    // ------------------------------------------------------------------
    // ALGORITHM TO PREVIOUS TARGET – TARGET SIDE
    // ------------------------------------------------------------------
    E_RobotState.AlgorithmPreviousTarget:
        yeControl    := RobotControl.vector;
        yinTargetMap := xinMapTarget;
        IF boVectorReached THEN
            eState := E_RobotState.DrivePoint5AlignRFID;//SwitchCoordinatesTarget;
        END_IF
 
    // ------------------------------------------------------------------
    // SWITCH COORDINATES – TARGET SIDE
    // Load target station coordinate from array, switch to position mode.
    // ------------------------------------------------------------------
    E_RobotState.SwitchCoordinatesTarget:
        yeControl                  := RobotControl.position;
		ystTargetPosition.reX      := REAL_TO_LREAL(xarstCoordinates[xinRfidTargetIndex].rePosX) + (crePreTargetDistance * xinTargetDirectionIndex);
        ystTargetPosition.reY      := REAL_TO_LREAL(xarstCoordinates[xinRfidTargetIndex].rePosY);
        ystTargetPosition.reWinkel := REAL_TO_LREAL(xarstCoordinates[xinRfidTargetIndex].reWinkel);
        IF boPositionReached THEN
            eState := E_RobotState.DrivePoint5AlignRFID;
        END_IF
 
    // ------------------------------------------------------------------
    // DRIVE TO POINT 5 – RFID ALIGNMENT POINT + ALIGN
    // Load RFID target coordinate before transitioning.
    // ------------------------------------------------------------------
    E_RobotState.DrivePoint5AlignRFID:
        yeControl := RobotControl.position;
		ystTargetPosition.reX      := REAL_TO_LREAL(xarstCoordinates[xinRfidTargetIndex].rePosX);
        ystTargetPosition.reY      := REAL_TO_LREAL(xarstCoordinates[xinRfidTargetIndex].rePosY);
        ystTargetPosition.reWinkel := REAL_TO_LREAL(xarstCoordinates[xinRfidTargetIndex].reWinkel);
        IF boPositionReached THEN
            eState := E_RobotState.DrivePoint6AtRFID;
        END_IF
 
    // ------------------------------------------------------------------
    // DRIVE TO POINT 6 – AT RFID SENSOR + ALIGN
    // ------------------------------------------------------------------
    E_RobotState.DrivePoint6AtRFID:
        yeControl := RobotControl.position;
        IF TRUE THEN
            eState := E_RobotState.ScanRFIDTarget;
        END_IF
 
    // ------------------------------------------------------------------
    // SCAN RFID – TARGET
    // Signal "waiting for RFID in" to controller. Wait for boRFIDComplete.
    // ------------------------------------------------------------------
    E_RobotState.ScanRFIDTarget:
        yeControl := RobotControl.idle;
        ystMqttOut.sJobState.boWaitForRfidIn := TRUE;
        IF boRfidComplete THEN
            ystMqttOut.sJobState.boWaitForRfidIn := FALSE;
            eState := E_RobotState.DrivePoint5;
        END_IF
 
    // ------------------------------------------------------------------
    // DRIVE TO POINT 5 + ALIGN (return from RFID sensor)
    // ------------------------------------------------------------------
    E_RobotState.DrivePoint5:
		yeControl := RobotControl.vector;
		yboDriveAway := TRUE;
        (*yeControl := RobotControl.position;
		ystTargetPosition.reX      := REAL_TO_LREAL(xarstCoordinates[xinRfidTargetIndex].rePosX) + (crePreTargetDistance * xinTargetDirectionIndex);
        ystTargetPosition.reY      := REAL_TO_LREAL(xarstCoordinates[xinRfidTargetIndex].rePosY);
        ystTargetPosition.reWinkel := REAL_TO_LREAL(xarstCoordinates[xinRfidTargetIndex].reWinkel);*)
        IF xboAwayFromObstacle THEN
			yboDriveAway := FALSE;
            eState := E_RobotState.DrivePoint9Drop;//DrivePoint8BeforeDrop;
        END_IF
 
    // ------------------------------------------------------------------
    // DRIVE TO POINT 8 – BEFORE DROP-OFF
    // ------------------------------------------------------------------
//     E_RobotState.DrivePoint8BeforeDrop:
//         yeControl := RobotControl.position;
// 		ystTargetPosition.reX      := REAL_TO_LREAL(xarstCoordinates[xinTargetIndex].rePosX) + (crePreTargetDistance * xinTargetDirectionIndex);
//         ystTargetPosition.reY      := REAL_TO_LREAL(xarstCoordinates[xinTargetIndex].rePosY);
//         ystTargetPosition.reWinkel := REAL_TO_LREAL(xarstCoordinates[xinTargetIndex].reWinkel);
//         IF boPositionReached THEN
//             eState := E_RobotState.DrivePoint9Drop;
//         END_IF
 
    // ------------------------------------------------------------------
    // DRIVE TO POINT 9 – DROP-OFF POSITION
    // ------------------------------------------------------------------
    E_RobotState.DrivePoint9Drop:
        yeControl := RobotControl.position;
		ystTargetPosition.reX      := REAL_TO_LREAL(xarstCoordinates[xinTargetIndex].rePosX);
        ystTargetPosition.reY      := REAL_TO_LREAL(xarstCoordinates[xinTargetIndex].rePosY);
        ystTargetPosition.reWinkel := REAL_TO_LREAL(xarstCoordinates[xinTargetIndex].reWinkel);
        IF boPositionReached THEN
            eState := E_RobotState.OpenGripper;
        END_IF
 
    // ------------------------------------------------------------------
    // OPEN GRIPPER
    // Wait for workpiece-released confirmation (boWorkpieceLoaded = FALSE).
    // ------------------------------------------------------------------
    E_RobotState.OpenGripper:
        yeControl := RobotControl.idle;
		Gripper.closeGripperCommand := FALSE;

		IF Gripper.state_out = CoreGripperControlState.Open THEN
			ystMqttOut.sJobState.boTransportWorkpiece := FALSE;
			ystMqttOut.sJobState.boWorkpiecePlaced    := TRUE;
			eState := E_RobotState.DrivePoint8AfterDrop;
// 		ELSIF TONGripperTime.Q THEN			// Backup, falls Gripper nicht öffnet	--------------------------------------------------------------------------------------------------------------------------------------Hier einmal
// 			eState := E_RobotState.Standby;	// Hier noch in sinnvolleren Zustand springen
	 	END_IF
 
    // ------------------------------------------------------------------
    // DRIVE TO POINT 8 – RETURN AFTER DROP-OFF
    // ------------------------------------------------------------------
    E_RobotState.DrivePoint8AfterDrop:
		yeControl := RobotControl.vector;
		yboDriveAway := TRUE;
       (* yeControl := RobotControl.position;
		ystTargetPosition.reX      := REAL_TO_LREAL(xarstCoordinates[xinTargetIndex].rePosX) + (crePreTargetDistance * xinTargetDirectionIndex);
        ystTargetPosition.reY      := REAL_TO_LREAL(xarstCoordinates[xinTargetIndex].rePosY);
        ystTargetPosition.reWinkel := REAL_TO_LREAL(xarstCoordinates[xinTargetIndex].reWinkel);
		ystMqttOut.sJobState.boWorkpiecePlaced    := FALSE;*)
        IF xboAwayFromObstacle THEN
			yboDriveAway := FALSE;
            eState := E_RobotState.SelectMapParkPosition;
			 yinTargetMap               := xinMapParking;
        END_IF
 
    // ------------------------------------------------------------------
    // SELECT MAP – PARKING POSITION
    // Start vector algorithm to parking. Output job-done signal.
    // Branch A: new job received while returning → CheckConfirmJob
    // Branch B: normal end                       → Standby
    // ------------------------------------------------------------------
    E_RobotState.SelectMapParkPosition:
		yboPassiveWait := FALSE;
		yboDriveAway := FALSE;
         yinTargetMap               := xinMapParking;
        yeControl                  := RobotControl.vector;
		IF eStateOld <> E_RobotState.DrivePoint1NoWorkpiece THEN
		ystMqttOut.sGeneralState.boReady := TRUE;
		END_IF
		IF xreDistFromGoal > creDistanzForTokenRelease  THEN
			ystMqttOut.sToken.boTokenRelease := TRUE;
		END_IF
        IF boVectorReached THEN
			eState := E_RobotState.Standby;
         ELSIF boNewJob THEN
                eState := E_RobotState.CheckConfirmJob;
		END_IF;
		
END_CASE
 {endregion}

TONTokenRequestTime(IN :=  (E_RobotState.WaitPassiveSource = eState) OR (E_RobotState.WaitpointReachedTarget = eState) ,PT := T#0.2S);
TONGripperTime(IN := (eState = E_RobotState.CloseGripper) OR (E_RobotState.OpenGripper = eState), PT := ctiGripperTime);
TONChargingDelay(IN := boCancelCharging, PT := T#3S);

END_IF
	
	//TEST FÜR PASSIVE WAIT
	//eState := E_RobotState.WaitPassiveTarget;
// ---------------------------------------------------------------------------
// Mirror active state to diagnostic output
// ---------------------------------------------------------------------------
yeCurrentState := eState;
 
{endregion}
{region 'old'}
// ---------------------------------------------------------------------------
// Global control output overrides by state group
// (same pattern as FB_StatesTest – set yeControl after CASE to guarantee
//  correct value regardless of internal state transitions within one scan)
// ---------------------------------------------------------------------------
 (*
// Vector states
IF  (eState = E_RobotState.SelectMapStart)
 OR (eState = E_RobotState.WaitpointReachedSource)
 OR (eState = E_RobotState.AlgorithmPreviousSource)
 OR (eState = E_RobotState.SelectMapTarget)
 OR (eState = E_RobotState.WaitpointReachedTarget)
 OR (eState = E_RobotState.AlgorithmPreviousTarget)
 OR (eState = E_RobotState.SelectMapParkPosition) THEN
    yeControl := RobotControl.vector;
END_IF
 
// Position states
IF  (eState = E_RobotState.SwitchCoordinatesSource)
 OR (eState = E_RobotState.DrivePoint1Align)
 OR (eState = E_RobotState.DrivePoint2Align)
 OR (eState = E_RobotState.AtChargingStation)
 OR (eState = E_RobotState.DrivePoint1AfterCharge)
 OR (eState = E_RobotState.AtStation)
 OR (eState = E_RobotState.DrivePoint1WithWorkpiece)
 OR (eState = E_RobotState.DrivePoint1NoWorkpiece)
 OR (eState = E_RobotState.DrivePoint3Align)
 OR (eState = E_RobotState.DrivePoint4)
 OR (eState = E_RobotState.ScanRFIDSource)
 OR (eState = E_RobotState.DrivePoint3ToTarget)
 OR (eState = E_RobotState.SwitchCoordinatesTarget)
 OR (eState = E_RobotState.DrivePoint5AlignRFID)
 OR (eState = E_RobotState.DrivePoint6AtRFID)
 OR (eState = E_RobotState.ScanRFIDTarget)
 OR (eState = E_RobotState.DrivePoint5)
 OR (eState = E_RobotState.DrivePoint8BeforeDrop)
 OR (eState = E_RobotState.DrivePoint9Drop)
 OR (eState = E_RobotState.DrivePoint8AfterDrop) THEN
    yeControl := RobotControl.position;
END_IF
 
// Idle states
IF  (eState = E_RobotState.LoadMaps)
 OR (eState = E_RobotState.Standby)
 OR (eState = E_RobotState.CloseGripper)
 OR (eState = E_RobotState.OpenGripper)
 OR (eState = E_RobotState.WaitForChargingDone) THEN
    yeControl := RobotControl.idle;
END_IF
 
// Stop states
IF  (eState = E_RobotState.WaitPassiveSource)
 OR (eState = E_RobotState.WaitPassiveTarget) THEN
    yeControl := RobotControl.stop;
END_IF*)
{endregion}

END_FUNCTION_BLOCK

// ---- POUs/HAWinoCore/01_Motors/Gripper.TcPOU
PROGRAM Gripper
VAR_INPUT
	closeGripperCommand		 : BOOL;
	Grippercurrent AT %I* : UINT;
END_VAR
VAR_OUTPUT
	state_out : CoreGripperControlState := CoreGripperControlState.init;
END_VAR
VAR
	state : CoreGripperControlState := CoreGripperControlState.init;
	slider					AT%I* : BOOL;
	partGripped				AT%I* : BOOL;
	
	driveEnable				AT%Q* : BOOL;
	driveVelocity 			AT%Q* : INT;
	current :INT;
	timer : TON;
	
	movementTime : TIME := T#3000MS; //Timevalue for Grippercurrent
END_VAR


current := UINT_TO_INT(Grippercurrent);

CASE state OF
///////////////////////////////////////////////////////////////
 CoreGripperControlState.Init: //Reference opening-drive 
 	state := CoreGripperControlState.opening;
			timer(in := 0, pt:= movementTime); // starts Timer
///////////////////////////////////////////////////////////////		
	CoreGripperControlState.Opening:
		driveEnable:=1;
		driveVelocity:=32767;
		IF current > 50 THEN
			timer(IN:=1);
		END_IF;
		
		IF timer.Q THEN 
			state := CoreGripperControlState.Open;
		END_IF
		state_out := CoreGripperControlState.Opening;
///////////////////////////////////////////////////////////////		
	CoreGripperControlState.Closing:
		driveEnable:=1;
		driveVelocity:=-32767;
		timer(IN:=1);
		IF timer.Q THEN 
			state := CoreGripperControlState.Closed;
		END_IF
		state_out := CoreGripperControlState.Closing;
		
///////////////////////////////////////////////////////////////	
	CoreGripperControlState.Open:	
		driveEnable:=0;
		driveVelocity:=0;
		IF  closeGripperCommand THEN
			state := CoreGripperControlState.Closing;
			timer(in := 0, pt:= movementTime);
		END_IF
		state_out := CoreGripperControlState.Open;
///////////////////////////////////////////////////////////////		
	CoreGripperControlState.Closed:	
		driveEnable:=1;
		driveVelocity:=0;					
		IF NOT closeGripperCommand THEN
			state := CoreGripperControlState.Opening;
			timer(in := 0, pt:= movementTime);
		END_IF
		state_out := CoreGripperControlState.Closed;
		
END_CASE

END_PROGRAM

// ---- POUs/HAWinoCore/05_Bahnplanung/FB_Mapping.TcPOU
FUNCTION_BLOCK FB_Mapping
VAR_INPUT
    xstMqttIn               : sMqttIn;  // Full MQTT input – sJOB.inDestination1/2 are read here
    xinDefaultParkingIndex  : INT;      // Constant parking index (e.g. IDX_PARKING_101)
                                        // passed straight through to output unchanged
END_VAR
 
VAR_OUTPUT
    // --- Indices for FB_RobotStateMachine ---
    yinSourceIndex          : INT;      // xinSourceIndex  of FB_RobotStateMachine
	yinSourceDirectionIndex : INT;      //1 if + and -1 if -
	yinTargetDirectionIndex : INT;      //1 if + and -1 if -
    yinTargetIndex          : INT;      // xinTargetIndex  of FB_RobotStateMachine
    yinRfidSourceIndex      : INT;      // xinRfidSourceIndex
    yinRfidTargetIndex      : INT;      // xinRfidTargetIndex
    yinParkingIndex         : INT;      // xinParkingIndex  (= xinDefaultParkingIndex, passed through)
    yinChargingIndex        : INT;      // xinChargingIndex (only valid when yboJobCharging = TRUE)
    yinMapSource            : INT;      // xinMapSource     (map ID derived from station group)
    yinMapTarget            : INT;      // xinMapTarget     (map ID derived from station group)
 
    // --- Job type flags ---
    yboJobTransport         : BOOL;     // Normal transport job  (D2 ≠ 404)
    yboJobCharging          : BOOL;     // Charging job          (D2 = 404)
    yboDecodeError          : BOOL;     // TRUE if an unknown station number was received
END_VAR
 
VAR
    inDest1                 : INT;      // Local copy of inDestination1
    inDest2                 : INT;      // Local copy of inDestination2
	RobotIndex: INT;
END_VAR

//   Station numbers and their RFID assignments:
//   ┌──────────┬────────────────────────┬───────────────────────────────────┐
//   │ Station  │ Name                   │ Associated RFID index             │
//   ├──────────┼────────────────────────┼───────────────────────────────────┤
//   │  1,  2   │ Storage  (left side)   │ RFID 1 (source) / RFID 2 (target) │
//   │  3,  4   │ Storage  (right side)  │ RFID 2 (source) / RFID 1 (target) │
//   │ 11, 12   │ Production 1+2 left    │ RFID 3 (source) / RFID 4 (target) │
//   │ 21, 22   │ Production 1+2 right   │ RFID 4 (source) / RFID 3 (target) │
//   │ 31, 32   │ Production 3+4 left    │ RFID 5 (source) / RFID 6 (target) │
//   │ 41, 42   │ Production 3+4 right   │ RFID 6 (source) / RFID 5 (target) │
//   │  5,  6   │ Drop-off  (left side)  │ RFID 7 (source) / RFID 8 (target) │
//   │  7,  8   │ Drop-off  (right side) │ RFID 8 (source) / RFID 7 (target) │
//   │201, 202  │ Charging               │ No RFID                            │
//   │101..104  │ Parking (constant)     │ No RFID                            │
//   └──────────┴────────────────────────┴───────────────────────────────────┘
// ---------------------------------------------------------------------------
// Reset outputs each scan
// ---------------------------------------------------------------------------
yinSourceIndex      := 0;
yinTargetIndex      := 0;
yinRfidSourceIndex  := IDX_RFID_1;
yinRfidTargetIndex  := IDX_RFID_1;
yinParkingIndex     := xinDefaultParkingIndex;
yinChargingIndex    := IDX_CHARGING_201;
yinMapSource        := 0;
yinMapTarget        := 0;
yboJobTransport     := FALSE;
yboJobCharging      := FALSE;
yboDecodeError      := FALSE;
 
// ---------------------------------------------------------------------------
// Read destinations from MQTT job struct
// ---------------------------------------------------------------------------
inDest1 := xstMqttIn.sJOB.inDestination1;
inDest2 := xstMqttIn.sJOB.inDestination2;
 
// ---------------------------------------------------------------------------
// Determine job type
// ---------------------------------------------------------------------------
IF inDest2 = 404 THEN
    yboJobCharging  := TRUE;
    yboJobTransport := FALSE;
ELSE
    yboJobCharging  := FALSE;
    yboJobTransport := TRUE;
END_IF
 
// ---------------------------------------------------------------------------
// DECODE SOURCE (Destination 1)
//
// Each station number maps to:
//   - a coordinate array index  (yinSourceIndex)
//   - the RFID index on the SOURCE side of that station (yinRfidSourceIndex)
//   - a map ID for the vector algorithm             (yinMapSource)
// ---------------------------------------------------------------------------
CASE inDest1 OF
 
    // --- Storage – left approach (stations 1, 2) ---
    1:
        yinSourceIndex     := IDX_STORAGE_1;
        yinRfidSourceIndex := IDX_RFID_1;
        yinMapSource       := 1;
		yinSourceDirectionIndex := -1;
 		
    2:
        yinSourceIndex     := IDX_STORAGE_2;
        yinRfidSourceIndex := IDX_RFID_1;
        yinMapSource       := 1;
 		yinSourceDirectionIndex := -1;
    // --- Storage – right approach (stations 3, 4) ---
    3:
        yinSourceIndex     := IDX_STORAGE_3;
        yinRfidSourceIndex := IDX_RFID_2;
        yinMapSource       := 2;
 		yinSourceDirectionIndex := 1;
 
    4:
        yinSourceIndex     := IDX_STORAGE_4;
        yinRfidSourceIndex := IDX_RFID_2;
        yinMapSource       := 2;
  		yinSourceDirectionIndex := 1;
 
    // --- Production 1+2 – left approach (stations 11, 12) ---
    11:
        yinSourceIndex     := IDX_PROD_11;
        yinRfidSourceIndex := IDX_RFID_3;
        yinMapSource       := 3;
 		yinSourceDirectionIndex := -1;
 
    12:
        yinSourceIndex     := IDX_PROD_12;
        yinRfidSourceIndex := IDX_RFID_3;
        yinMapSource       := 3;
 		yinSourceDirectionIndex := -1;
 
    // --- Production 1+2 – right approach (stations 21, 22) ---
    21:
        yinSourceIndex     := IDX_PROD_21;
        yinRfidSourceIndex := IDX_RFID_4;
        yinMapSource       := 4;
  		yinSourceDirectionIndex := 1;
 
    22:
        yinSourceIndex     := IDX_PROD_22;
        yinRfidSourceIndex := IDX_RFID_4;
        yinMapSource       := 4;
  		yinSourceDirectionIndex := 1;
 
    // --- Production 3+4 – left approach (stations 31, 32) ---
    31:
        yinSourceIndex     := IDX_PROD_31;
        yinRfidSourceIndex := IDX_RFID_5;
        yinMapSource       := 5;
 		yinSourceDirectionIndex := -1;
 
    32:
        yinSourceIndex     := IDX_PROD_32;
        yinRfidSourceIndex := IDX_RFID_5;
        yinMapSource       := 5;
 		yinSourceDirectionIndex := -1;
 
    // --- Production 3+4 – right approach (stations 41, 42) ---
    41:
        yinSourceIndex     := IDX_PROD_41;
        yinRfidSourceIndex := IDX_RFID_6;
        yinMapSource       := 6;
  		yinSourceDirectionIndex := 1;
 
    42:
        yinSourceIndex     := IDX_PROD_42;
        yinRfidSourceIndex := IDX_RFID_6;
        yinMapSource       := 6;
  		yinSourceDirectionIndex := 1;
 
    // --- Drop-off – left approach (stations 5, 6) ---
    5:
        yinSourceIndex     := IDX_DROPOFF_5;
        yinRfidSourceIndex := IDX_RFID_7;
        yinMapSource       := 7;
 		yinSourceDirectionIndex := -1;
 
    6:
        yinSourceIndex     := IDX_DROPOFF_6;
        yinRfidSourceIndex := IDX_RFID_7;
        yinMapSource       := 7;
 		yinSourceDirectionIndex := -1;
 
    // --- Drop-off – right approach (stations 7, 8) ---
    7:
        yinSourceIndex     := IDX_DROPOFF_7;
        yinRfidSourceIndex := IDX_RFID_8;
        yinMapSource       := 8;
  		yinSourceDirectionIndex := 1;
 
    8:
        yinSourceIndex     := IDX_DROPOFF_8;
        yinRfidSourceIndex := IDX_RFID_8;
        yinMapSource       := 8;
  		yinSourceDirectionIndex := 1;
 
    // --- Charging stations (Destination1 = charging means the robot should charge) ---
    201:
        yinSourceIndex   := IDX_CHARGING_201;
        yinChargingIndex := IDX_CHARGING_201;
        yinMapSource     := 9;
 
    202:
        yinSourceIndex   := IDX_CHARGING_202;
        yinChargingIndex := IDX_CHARGING_202;
        yinMapSource     := 9;
 
ELSE
    // Unknown station number
    yboDecodeError := TRUE;
 
END_CASE
 
// ---------------------------------------------------------------------------
// DECODE TARGET (Destination 2)
//
// Each station number maps to:
//   - a coordinate array index  (yinTargetIndex)
//   - the RFID index on the TARGET side of that station (yinRfidTargetIndex)
//   - a map ID for the vector algorithm             (yinMapTarget)
//
// Special case: Destination2 = 404 → charging job, no target station needed.
// The RFID on the TARGET side is the opposite side of the same block:
//   left stations  (1,2 / 11,12 / 31,32 / 5,6)  → approached from the right → RFID 2,4,6,8
//   right stations (3,4 / 21,22 / 41,42 / 7,8)  → approached from the left  → RFID 1,3,5,7
// ---------------------------------------------------------------------------
CASE inDest2 OF
 
    // --- Storage – right approach as TARGET (stations 1, 2) ---
    1:
        yinTargetIndex     := IDX_STORAGE_1;
        yinRfidTargetIndex := IDX_RFID_1;
        yinMapTarget       := 1;
  		yinTargetDirectionIndex := -1;
 
    2:
        yinTargetIndex     := IDX_STORAGE_2;
        yinRfidTargetIndex := IDX_RFID_1;
        yinMapTarget       := 1;
   		yinTargetDirectionIndex := -1;
 
    // --- Storage – left approach as TARGET (stations 3, 4) ---
    3:
        yinTargetIndex     := IDX_STORAGE_3;
        yinRfidTargetIndex := IDX_RFID_2;
        yinMapTarget       := 2;
   		yinTargetDirectionIndex := 1;
 
    4:
        yinTargetIndex     := IDX_STORAGE_4;
        yinRfidTargetIndex := IDX_RFID_2;
        yinMapTarget       := 2;
   		yinTargetDirectionIndex := 1;
 
    // --- Production 1+2 – right approach as TARGET (stations 11, 12) ---
    11:
        yinTargetIndex     := IDX_PROD_11;
        yinRfidTargetIndex := IDX_RFID_3;
        yinMapTarget       := 3;
   		yinTargetDirectionIndex := -1;
 
    12:
        yinTargetIndex     := IDX_PROD_12;
        yinRfidTargetIndex := IDX_RFID_3;
        yinMapTarget       := 3;
   		yinTargetDirectionIndex := -1;
 
    // --- Production 1+2 – left approach as TARGET (stations 21, 22) ---
    21:
        yinTargetIndex     := IDX_PROD_21;
        yinRfidTargetIndex := IDX_RFID_4;
        yinMapTarget       := 4;
   		yinTargetDirectionIndex := 1;
 
    22:
        yinTargetIndex     := IDX_PROD_22;
        yinRfidTargetIndex := IDX_RFID_4;
        yinMapTarget       := 4;
   		yinTargetDirectionIndex := 1;
 
    // --- Production 3+4 – right approach as TARGET (stations 31, 32) ---
    31:
        yinTargetIndex     := IDX_PROD_31;
        yinRfidTargetIndex := IDX_RFID_5;
        yinMapTarget       := 5;
   		yinTargetDirectionIndex := -1;
 
    32:
        yinTargetIndex     := IDX_PROD_32;
        yinRfidTargetIndex := IDX_RFID_5;
        yinMapTarget       := 5;
   		yinTargetDirectionIndex := -1;
 
    // --- Production 3+4 – left approach as TARGET (stations 41, 42) ---
    41:
        yinTargetIndex     := IDX_PROD_41;
        yinRfidTargetIndex := IDX_RFID_6;
        yinMapTarget       := 6;
		yinTargetDirectionIndex := 1;
 
    42:
        yinTargetIndex     := IDX_PROD_42;
        yinRfidTargetIndex := IDX_RFID_6;
        yinMapTarget       := 6;
		yinTargetDirectionIndex := 1;
 
    // --- Drop-off – right approach as TARGET (stations 5, 6) ---
    5:
        yinTargetIndex     := IDX_DROPOFF_5;
        yinRfidTargetIndex := IDX_RFID_7;
        yinMapTarget       := 7;
   		yinTargetDirectionIndex := -1;
 
    6:
        yinTargetIndex     := IDX_DROPOFF_6;
        yinRfidTargetIndex := IDX_RFID_7;
        yinMapTarget       := 7;
   		yinTargetDirectionIndex := -1;
 
    // --- Drop-off – left approach as TARGET (stations 7, 8) ---
    7:
        yinTargetIndex     := IDX_DROPOFF_7;
        yinRfidTargetIndex := IDX_RFID_8;
        yinMapTarget       := 8;
   		yinTargetDirectionIndex := 1;
 
    8:
        yinTargetIndex     := IDX_DROPOFF_8;
        yinRfidTargetIndex := IDX_RFID_8;
        yinMapTarget       := 8;
   		yinTargetDirectionIndex := 1;
		
    // --- Special: charging job (Destination2 = 404) ---
    404:
        // Target indices not relevant for charging – leave at default.
        // yboJobCharging is already TRUE from the job-type block above.
        yinTargetIndex     := yinChargingIndex;
        yinRfidTargetIndex := IDX_RFID_1;   // unused for charging
        yinMapTarget       := 9;
 
ELSE
    // Unknown target station number (only flag error if not a charging job)
    IF NOT yboJobCharging THEN
        yboDecodeError := TRUE;
    END_IF
 
END_CASE
 
// ---------------------------------------------------------------------------
// Parking index is always passed through unchanged
// ---------------------------------------------------------------------------
RobotIndex := Var_HAWIno.Robot_Number;
 CASE RobotIndex OF 
	1:yinParkingIndex := IDX_PARKING_101;
	2:yinParkingIndex := IDX_PARKING_102;
	3:yinParkingIndex := IDX_PARKING_103;
	4:yinParkingIndex := IDX_PARKING_104;
END_CASE

END_FUNCTION_BLOCK

// ---- POUs/HAWinoCore/05_Bahnplanung/FB_MQTT.TcPOU
FUNCTION_BLOCK FB_MQTT
VAR
    fbClient        : FB_IotMqttClient;
    fbMessageQueue  : FB_IotMqttMessageQueue;
    fbMessage       : FB_IotMqttMessage;
    bSubscribed     : BOOL;
    sReceived       : STRING;
    bSendError   : BOOL;
	bSendJob	:	BOOL;
	bSendState	: BOOL;
	bSendToken	: BOOL;
    sReceivedjob	: STRING(1000);
	sReceivedcmd 	: STRING(1000);
	sSendError    : STRING(1000);
	sSendJob    : STRING(1000);
	sSendState    : STRING := 'State';
	sSendToken    : STRING := 'Token';
	sMqttSEND : sMqttOut;
	sMqttRECEIVE : sMqttIn;
	sSendCharging : STRING;
	
	//Alten Strings speichern
	tempsSendError : STRING(1000);
	tempsSendJob : STRING(1000);
	tempsSendState : STRING(1000);
	tempsSendToken : STRING(1000);
	
	    // JSON Parser
    fbJson          : FB_JsonDomParser;
    jsonDoc         : SJsonValue;
    jsonNode        : SJsonValue;
    
    // Parsed Variablen Empfangen
    boStop          : BOOL;
    boReset         : BOOL;
    boJobReset      : BOOL;
	boRfidComplete	: BOOL;
	boStartJob		: BOOL;
	boTokenGrant	: BOOL;
	boCancelCharging: BOOL;
	
	// Parsed Variablen Senden
	boErrorRoutePlanning: BOOL := FALSE;
	boErrorControl		: BOOL := FALSE;
	boErrorNoWorkpiece	:BOOL := FALSE;
	boErrorWorkpieceLost: BOOL := FALSE;
	
	//Brauchte ne VAR
	charging_dock : INT;
	loading_speed : INT;
	sSendStop : STRING;
	tempjob : STRING;
	tempcmd : STRING;
	tempserror : STRING;
	tempsjob : STRING;
	tempsstate : STRING;
	tempstoken : STRING;
	start : BOOL;
	sReceivedStart : STRING;
	LADEN : BOOL;
	TONPosition : TON;
	boTONFlanke : BOOL;
	tempInit : STRING;
	temprToken : STRING;
	sReceivedToken : STRING;
	station_id : STRING;
	
END_VAR

VAR_INPUT
	xsDataToSend : sMqttOut;
	xsKoordinate : sKoordinate;
	xinMqttTokenTargetId : INT;
END_VAR
VAR_OUTPUT
	ysDataToReceive : sMqttIn;
END_VAR

// Verbindungsparameter setzen

fbClient.sHostName	:=	'192.168.0.11';
fbClient.nHostPort	:= 	1883;
fbClient.sUserName	:=	'VPJ';
fbClient.sUserPassword	:=	'R462';

// Queue mit Client verknüpfen
fbClient.ipMessageQueue := fbMessageQueue;
fbClient.Execute(bConnect := TRUE);

sMqttSEND := xsDataToSend;

// Einmalig subscriben wenn verbunden
IF fbClient.bConnected AND NOT bSubscribed THEN
	tempjob := CONCAT('HAWino/', INT_TO_STRING(Robot_Number));
	tempjob := CONCAT(tempjob, '/job');
    fbClient.Subscribe(
        sTopic := tempjob,
        eQoS   := 0
    );
	tempcmd := CONCAT('HAWino/', INT_TO_STRING(Robot_Number));
	tempcmd := CONCAT(tempcmd, '/cmd');
	fbClient.Subscribe(
        sTopic := tempcmd,
        eQoS   := 0
    );
	
	tempInit := CONCAT('HAWino/', INT_TO_STRING(Robot_Number));
	tempInit := CONCAT(tempInit, '/init');
	fbClient.Subscribe(
        sTopic := tempInit,
        eQoS   := 0
    );
	
	temprToken := CONCAT('HAWino/', INT_TO_STRING(Robot_Number));
	temprToken := CONCAT(temprToken, '/token');
	fbClient.Subscribe(
        sTopic := temprToken,
        eQoS   := 0
    );
	
	tempserror := CONCAT('HAWino/', INT_TO_STRING(Robot_Number));
	tempserror := CONCAT(tempserror, '/error');
	
	tempsjob := CONCAT('HAWino/', INT_TO_STRING(Robot_Number));
	tempsjob := CONCAT(tempsjob, '/jobState');
	
	tempsstate := CONCAT('HAWino/', INT_TO_STRING(Robot_Number));
	tempsstate := CONCAT(tempsstate, '/generalState');
	
// 	tempstoken := CONCAT('agents/station/test_station/token', INT_TO_STRING(Robot_Number));
// 	tempstoken := CONCAT(tempstoken, '/token');
	
	bSubscribed := TRUE;
END_IF

// Nachrichten aus Queue lesen
IF fbMessageQueue.nQueuedMessages > 0 THEN
    fbMessageQueue.Dequeue(fbMessage := fbMessage);
    fbMessage.GetPayload(
        pPayload             := ADR(sReceived),
        nPayloadSize         := SIZEOF(sReceived),
        bSetNullTermination  := TRUE
    );
	    IF fbMessage.CompareTopic(sTopic := tempjob) THEN
        fbMessage.GetPayload(pPayload := ADR(sReceivedjob), nPayloadSize := SIZEOF(sReceivedjob), bSetNullTermination := TRUE);
    
    	ELSIF fbMessage.CompareTopic(sTopic := tempcmd) THEN
        fbMessage.GetPayload(pPayload := ADR(sReceivedcmd), nPayloadSize := SIZEOF(sReceivedcmd), bSetNullTermination := TRUE);
		
 		ELSIF fbMessage.CompareTopic(sTopic := tempInit) THEN
         fbMessage.GetPayload(pPayload := ADR(sReceivedStart), nPayloadSize := SIZEOF(sReceivedStart), bSetNullTermination := TRUE);
 		ELSIF fbMessage.CompareTopic(sTopic := temprToken) THEN
         fbMessage.GetPayload(pPayload := ADR(sReceivedToken), nPayloadSize := SIZEOF(sReceivedToken), bSetNullTermination := TRUE);
		END_IF
	
// Start Parsen
    // jsonDoc := fbJson.ParseDocument(sReceivedStart);
	
  (*   IF jsonDoc <> 0 THEN
         // Init auslesen
        jsonNode := fbJson.FindMember(jsonDoc, 'test');
         IF jsonNode <> 0 THEN
             start := fbJson.GetString(jsonNode) = 'TRUE';
         END_IF
	*)
	
	// JSON parsen CMD
    jsonDoc := fbJson.ParseDocument(sReceivedcmd);
    
    IF jsonDoc <> 0 THEN
        // boStop auslesen
        jsonNode := fbJson.FindMember(jsonDoc, 'boStop');
        IF jsonNode <> 0 THEN
            sMqttRECEIVE.sCmd.boStop := fbJson.GetBool(jsonNode);
        END_IF
        
        // boReset auslesen
        jsonNode := fbJson.FindMember(jsonDoc, 'boReset');
        IF jsonNode <> 0 THEN
            sMqttRECEIVE.sCmd.boReset := fbJson.GetBool(jsonNode);
        END_IF
        
        // boJobReset auslesen
        jsonNode := fbJson.FindMember(jsonDoc, 'boJobReset');
        IF jsonNode <> 0 THEN
            sMqttRECEIVE.sCmd.boJobReset := fbJson.GetBool(jsonNode);
        END_IF
		
		// boRfidComplete auslesen
        jsonNode := fbJson.FindMember(jsonDoc, 'boRfidComplete');
        IF jsonNode <> 0 THEN
            sMqttRECEIVE.sCmd.boRFIDComplete := fbJson.GetBool(jsonNode);
        END_IF
		
		// boStartJob auslesen
        jsonNode := fbJson.FindMember(jsonDoc, 'boStartJob');
        IF jsonNode <> 0 THEN
            sMqttRECEIVE.sCmd.boStartJob := fbJson.GetBool(jsonNode);
        END_IF
		
// 		// boTokenGrant auslesen
//         jsonNode := fbJson.FindMember(jsonDoc, 'boTokenGrant');
//         IF jsonNode <> 0 THEN
//             sMqttRECEIVE.sCmd.boTokenGrant := fbJson.GetString(jsonNode) = 'TRUE';
//         END_IF
		
		// boCancelCharging auslesen
        jsonNode := fbJson.FindMember(jsonDoc, 'boCancelCharging');
        IF jsonNode <> 0 THEN
            sMqttRECEIVE.sCmd.boCancelCharging := fbJson.GetBool(jsonNode);
        END_IF
    END_IF
	
	// JSON parsen CMD
    jsonDoc := fbJson.ParseDocument(sReceivedjob);
	
    IF jsonDoc <> 0 THEN
        // JobID auslesen
        jsonNode := fbJson.FindMember(jsonDoc, 'jobId');
        IF jsonNode <> 0 THEN
            sMqttRECEIVE.sJOB.inJobID := DINT_TO_INT(fbJson.GetInt(jsonNode));
        END_IF
        
        // Destination 1 auslesen
        jsonNode := fbJson.FindMember(jsonDoc, 'inDestination1');
        IF jsonNode <> 0 THEN
            sMqttRECEIVE.sJOB.inDestination1 := DINT_TO_INT(fbJson.GetInt(jsonNode));
        END_IF
        
        // Destination 2 auslesen
        jsonNode := fbJson.FindMember(jsonDoc, 'inDestination2');
        IF jsonNode <> 0 THEN
            sMqttRECEIVE.sJOB.inDestination2 := DINT_TO_INT(fbJson.GetInt(jsonNode));
        END_IF
    END_IF
	
	// JSON parsen Token
    jsonDoc := fbJson.ParseDocument(sReceivedToken);
    IF jsonDoc <> 0 THEN
        // Token Granted auslesen
		jsonNode := fbJson.FindMember(jsonDoc, 'category');
		IF jsonNode <> 0 THEN
			IF fbJson.GetString(jsonNode) = 'TOKEN_GRANT' THEN
				sMqttRECEIVE.sCmd.boTokenGrant := TRUE;
			END_IF
		END_IF
    END_IF
END_IF

start := TRUE;

IF start THEN
	// Die gesendeten Strings abspeichern
	tempsSendError := sSendError;
	tempsSendJob := sSendJob;
	tempsSendState := sSendState;
	tempsSendToken := sSendToken;
	
	
	// Kompletten Error-JSON zusammenbauen
	sSendError := CONCAT('{"boErrorRoutePlanning":"', BOOL_TO_STRING(sMqttSEND.sError.boErrorRoutePlanning));
	sSendError := CONCAT(sSendError, '","boErrorControl":"');
	sSendError := CONCAT(sSendError, BOOL_TO_STRING(sMqttSEND.sError.boErrorControl));
	sSendError := CONCAT(sSendError, '","boErrorNoWorkpiece":"');
	sSendError := CONCAT(sSendError, BOOL_TO_STRING(sMqttSEND.sError.boErrorNoWorkpiece));
	sSendError := CONCAT(sSendError, '","boErrorWorkpieceLost":"');
	sSendError := CONCAT(sSendError, BOOL_TO_STRING(sMqttSEND.sError.boErrorWorkpieceLost));
	sSendError := CONCAT(sSendError, '"}');
	
	// Kompletten jobState-JSON zusammenbauen
	sSendJob := CONCAT('{"boWorkpieceLoaded":"', BOOL_TO_STRING(sMqttSEND.sJobState.boWorkpieceLoaded));
	sSendJob := CONCAT(sSendJob, '","boTransportWorkpiece":"');
	sSendJob := CONCAT(sSendJob, BOOL_TO_STRING(sMqttSEND.sJobState.boTransportWorkpiece));
	sSendJob := CONCAT(sSendJob, '","boJobAccepted":"');
	sSendJob := CONCAT(sSendJob, BOOL_TO_STRING(sMqttSEND.sJobState.boJobAccepted));
	sSendJob := CONCAT(sSendJob, '","boWaitForRfidOut":"');
	sSendJob := CONCAT(sSendJob, BOOL_TO_STRING(sMqttSEND.sJobState.boWaitForRfidOut));
	sSendJob := CONCAT(sSendJob, '","boWaitForRfidIn":"');
	sSendJob := CONCAT(sSendJob, BOOL_TO_STRING(sMqttSEND.sJobState.boWaitForRfidIn));
	sSendJob := CONCAT(sSendJob, '","boWorkpiecePlaced":"');
	sSendJob := CONCAT(sSendJob, BOOL_TO_STRING(sMqttSEND.sJobState.boWorkpiecePlaced));
	sSendJob := CONCAT(sSendJob, '"}');
	
	
	sMqttSEND.sGeneralState.strPosition := CONCAT(CONCAT(REAL_TO_STRING(xsKoordinate.rePosX),','),REAL_TO_STRING(xsKoordinate.rePosY));
	
	// Kompletten generalState-JSON zusammenbauen
	sSendState := CONCAT('{"boReady":"', BOOL_TO_STRING(sMqttSEND.sGeneralState.boReady));
	sSendState := CONCAT(sSendState, '","boCharging":"');
	sSendState := CONCAT(sSendState, BOOL_TO_STRING(sMqttSEND.sGeneralState.boCharging));
	sSendState := CONCAT(sSendState, '","strPosition":"');
	sSendState := CONCAT(sSendState, sMqttSEND.sGeneralState.strPosition);
	sSendState := CONCAT(sSendState, '"}');
	
	// Kompletten Token-JSON
	IF sMqttSEND.sToken.boTokenRequest THEN
		sSendToken := CONCAT('{"category":"TOKEN_REQUEST","robot_id":"', INT_TO_STRING(Robot_Number));
		sSendToken := CONCAT(sSendToken, '"}');
	END_IF
	IF sMqttSEND.sToken.boTokenRelease THEN
		sSendToken := CONCAT('{"category":"TOKEN_RELEASE","robot_id":"', INT_TO_STRING(Robot_Number));
		sSendToken := CONCAT(sSendToken, '"}');
	END_IF
	
	//Charging Request
	sSendCharging := CONCAT('{"robot":"', INT_TO_STRING(Robot_Number));
	sSendCharging := CONCAT(sSendCharging, '","charge":"true');
	sSendCharging := CONCAT(sSendCharging, '","charging_dock":"');
	sSendCharging := CONCAT(sSendCharging, INT_TO_STRING(charging_dock));
	sSendCharging := CONCAT(sSendCharging, '","loading_speed":"');
	sSendCharging := CONCAT(sSendCharging, INT_TO_STRING(loading_speed));
	sSendCharging := CONCAT(sSendCharging, '"}');
	
	//Aufladen stoppen
	sSendStop := CONCAT('{"robot":"', INT_TO_STRING(Robot_Number));
	sSendStop := CONCAT(sSendStop, '","charge":"false');
	sSendStop := CONCAT(sSendStop, '","charging_dock":"');
	sSendStop := CONCAT(sSendStop, INT_TO_STRING(charging_dock));
	sSendStop := CONCAT(sSendStop, '","loading_speed":"');
	sSendStop := CONCAT(sSendStop, INT_TO_STRING(loading_speed));
	sSendStop := CONCAT(sSendStop, '"}');
	
	
	
	// Nur senden wenn sich etwas geändert hat
	IF tempsSendError <> sSendError THEN
		bSendError := TRUE;
	END_IF
	IF tempsSendJob <> sSendJob THEN
		bSendJob := TRUE;
	END_IF

	
	TONPosition(IN := NOT boTONFlanke ,PT := T#0.5S);
	boTONFlanke := TONPOsition.Q;	
	
	IF boTONFlanke THEN
		bSendState := TRUE;
	END_IF

	IF tempsSendToken <> sSendToken THEN
		bSendToken := TRUE;
	END_IF
	
	
	IF fbClient.bConnected THEN
		IF bSendError THEN
			fbClient.Publish(
				sTopic       := tempserror,
				pPayload     := ADR(sSendError),
				nPayloadSize := LEN(sSendError),
				eQoS         := 0,
				bRetain      := FALSE,
				bQueue       := FALSE
			);
			bSendError := FALSE;
		END_IF
	
		IF bSendJob THEN
			fbClient.Publish(
				sTopic       := tempsjob,
				pPayload     := ADR(sSendJob),
				nPayloadSize := LEN(sSendJob),
				eQoS         := 0,
				bRetain      := FALSE,
				bQueue       := FALSE
			);
			bSendJob := FALSE;
		END_IF
	
		IF bSendState THEN
			fbClient.Publish(
				sTopic       := tempsstate,
				pPayload     := ADR(sSendState),
				nPayloadSize := LEN(sSendState),
				eQoS         := 0,
				bRetain      := FALSE,
				bQueue       := FALSE
			);
			bSendState := FALSE;
		END_IF
	
	CASE xinMqttTokenTargetId OF
		1: station_id := 'storage_1';
		2: station_id := 'manufacturing_1';
		3: station_id := 'manufacturing_3';
		4: station_id := 'manufacturing_3';
		5: station_id := 'dispatch';
		
	END_CASE
	tempstoken := CONCAT('agents/station/', station_id); 
	tempstoken := CONCAT(tempstoken,'/token');
		IF bSendToken THEN
			fbClient.Publish(
				sTopic       := tempstoken,
				pPayload     := ADR(sSendToken),
				nPayloadSize := LEN(sSendToken),
				eQoS         := 0,
				bRetain      := FALSE,
				bQueue       := FALSE
			);
			bSendToken := FALSE;
		END_IF
// 		// Roboter will Laden
//  		IF NOT LADEN THEN
//   			fbClient.Publish(
//   				sTopic       := 'ChargingRequest',
//   				pPayload     := ADR(sSendCharging),
//   				nPayloadSize := LEN(sSendCharging),
//   				eQoS         := 0,
//   				bRetain      := FALSE,
//   				bQueue       := FALSE
//   			);
// 			LADEN		 := TRUE;
//  		END_IF
// 		//Roboter soll laden beenden
// 		IF boCancelCharging = TRUE AND E_RobotState = 8 THEN
// 			fbClient.Publish(
// 				sTopic       := 'ChargingRequest',
// 				pPayload     := ADR(sSendStop),
// 				nPayloadSize := LEN(sSendStop),
// 				eQoS         := 0,
// 				bRetain      := FALSE,
// 				bQueue       := FALSE
// 			);
// 		END_IF
	END_IF
END_IF

ysDataToReceive := sMqttRECEIVE;

END_FUNCTION_BLOCK

// ---- POUs/HAWinoCore/HAWino.TcPOU
PROGRAM HAWino
VAR
	Robot_Number	AT%Q*	: INT;
	operationState : DUT_SysState := DUT_SysState.init; 
	RobotData : RobotInternalData;
	GetId : Tc2_Utilities.FB_GetSystemId;
	init : INT;
	SysGUID : GUID;
	start : BOOL:= TRUE;
	
	// Outputs
	initDone AT%Q* : BOOL := FALSE;
	cameraPosition AT%Q* : Position := (x := 0.0, y := 0.0, theta := 0.0, e := 0.0);	// Aktuelle roboterspezifische Kameraposition
	cameraReceivedPakets AT%Q* : UINT;													// Counter für erhaltene Kamerapakete
END_VAR

CASE operationState OF
	//Get SysId for Identification
	DUT_SysState.init:
		GetId(bexecute := start,stSystemId=>SysGUID);
		IF NOT GetId.bBusy THEN	
			operationState:=DUT_SysState.preOp;
		END_IF
	DUT_SysState.preOp:
	//Set RobotNumber for MQTT and set flag to start MQTT
		IF InitSysId(GUID_to_String(SysGUID)) THEN
			Var_HAWIno.Robot_Number := RobotData.Robot_Number;		
			initDone := TRUE;
			operationState:=DUT_SysState.Op;
		END_IF
	DUT_SysState.Op:
	//Operate System

		MQTT();
		IrDistanceSensors();
		Camera();
		cameraPosition := Camera.cameraData.robotPosition[RobotData.Robot_Number]; //Zuweisung der roboterspezifischen Kameraposition
		cameraReceivedPakets := Camera.cameraData.nReceivedPakets;	// Zuweisung der Anzahl der vom Kamerasystem versendeten Pakete (Ueberwachungszwecke)
END_CASE

METHOD InitSysId : BOOL
VAR_INPUT
	SysId : STRING;
END_VAR
VAR
	state : INT;
	CX31C9D6 : STRING := '77726FC0-DD5E-F7D7-002E-41ED9B95AABA';
	CX35CFB8 : STRING := '2A7FC16A-555A-D05D-0E28-E804E05477FE';
	CX35CDC8 : STRING := 'AD3D576A-9CE4-FB95-7439-909C21AA2B33';
	CX35CDD6 : STRING := '975A6B25-37E2-0E46-4C4D-43CCC26F2A66';
	CX4D0046 : STRING := '4FFA7061-8E1F-E1C9-731A-38EAA9BAEAC6';
END_VAR
// CX-31C9D6 = 1
// CX-35CFB8 = 2
// CX-35CDC8 = 3
// CX-35CDD6 = 4
// CX-4D0046 = 5
IF SysId = CX31C9D6 THEN
	state := 1;
ELSIF SysId = CX35CFB8 THEN
	state := 2;
ELSIF SysId = CX35CDC8 THEN
	state := 3;
ELSIF SysId = CX35CDD6 THEN
	state := 4;
ELSIF SysId = CX4D0046 THEN
	state := 5;
ELSE
	state := 0;
END_IF

CASE state OF 
		1 : 	
				RobotData.Robot_IP_WiFi :='192.169.0.18';
				RobotData.Robot_IP_Wire :='192.169.0.28';
				RobotData.Robot_Name :='CX-35C9D6';
				RobotData.Robot_Nickname :='9D6';
				RobotData.Robot_Number := 1;
				RobotData.factor_V_m := 0.0361;
				RobotData.sum_V_b := -0.4916;
				RobotData.factor_I_m := 0;
				RobotData.sum_I_b := -0.13;
				InitSysId := TRUE;
				
				
		2:
				RobotData.Robot_IP_WiFi :='192.169.0.17';
				RobotData.Robot_IP_Wire :='192.169.0.27';
				RobotData.Robot_Name :='CX-35CFB8';
				RobotData.Robot_Nickname :='FB8';
				RobotData.Robot_Number := 2;
				RobotData.factor_V_m := 0.0315;
				RobotData.sum_V_b := -0.3835;
				RobotData.factor_I_m := 0;
				RobotData.sum_I_b := -0.045;
				InitSysId := TRUE;
		3:
				RobotData.Robot_IP_WiFi :='192.169.0.16';
				RobotData.Robot_IP_Wire :='192.169.0.26';
				RobotData.Robot_Name :='CX-35CDC8';
				RobotData.Robot_Nickname :='DC8';
				RobotData.Robot_Number := 3;
				RobotData.factor_V_m := 0.0350;
				RobotData.sum_V_b := -0.5301;
				RobotData.factor_I_m := 0;
				RobotData.sum_I_b := -0.08;
				InitSysId := TRUE;
		4:
				RobotData.Robot_IP_WiFi :='192.169.0.15';
				RobotData.Robot_IP_Wire :='192.169.0.25';
				RobotData.Robot_Name :='CX-35CDD6';
				RobotData.Robot_Nickname :='DD6';
				RobotData.Robot_Number := 4;
				RobotData.factor_V_m := 0.034;
				RobotData.sum_V_b := -0.404;
				RobotData.factor_I_m := 0;
				RobotData.sum_I_b := -0.08;
				InitSysId := TRUE;
		5:
				RobotData.Robot_IP_WiFi :='192.169.0.19';
				RobotData.Robot_IP_Wire :='192.169.0.29';
				RobotData.Robot_Name :='CX-04D0046';
				RobotData.Robot_Nickname :='046';
				RobotData.Robot_Number := 5;
				RobotData.factor_V_m := 0.0286;
				RobotData.sum_V_b := -0.2812;
				RobotData.factor_I_m := 0;
				RobotData.sum_I_b := 0;
				InitSysId := TRUE;			
		ELSE	//Ungültige Roboter Nummer
				RobotData.Robot_IP_WiFi :='0.0.0.0';
				RobotData.Robot_IP_Wire :='0.0.0.0';
				RobotData.Robot_Name :='Invalid';
				RobotData.Robot_Nickname :='Invalid';
				RobotData.Robot_Number := 0;
				InitSysId := false;
	END_CASE;
END_METHOD

END_PROGRAM

// ---- POUs/HAWinoCore/03_Communication/MQTT.TcPOU
PROGRAM MQTT
VAR
	fbIotMqttClient : FB_IotMqttClient;
    bSetParameter   : BOOL := TRUE;
    bConnect        : BOOL := TRUE;
	
	sTopicPub   	: STRING(255);
	sTopicPubAlive	: STRING(255);
    sPayloadPub 	: STRING(255);
	
	
    fbTimer : TON := (PT := T#1S); // Timer for LifeBit
	fbTimerPubPos : TON := (PT := T#20MS); // Timer for Publishing Position
	fbTimerPubSoC : TON := (PT := T#10S); // Timer for Publishing SoC
	fbTimerPubBat : TON := (PT := T#5S); // Timer for Battery Data
	
	(* received message *)
	
    bSubscribed    : BOOL;
    sTopicSub      : STRING(255);
    sTopicRcv      : STRING(255);
   
    sPayloadRcv    : STRING(255);
    fbMessageQueue : FB_IotMqttMessageQueue;
    fbMessage      : FB_IotMqttMessage;
	
	User : STRING := 'VPJ';
	Password : STRING := 'R462';
	IPAdress : STRING := '192.168.0.11';
	HostPort : UINT := 1883;
	
	sPayloadRcv1 : STRING(255);
    sPayloadRcv2 : STRING(255);
	
	sTopicSubJob : STRING(255) ;
	
	// **POSITION CODE**
	sTopicPubToRobotPosition : STRING(255); 
	bSubscribedPos : STRING(255);
	sTopicSubPos : STRING(255);
	robotPositionTopic : STRING;
	
	livePosition AT %I*: Position; 	// aktuelle Roboterposition vom Beobachter
	XKoordinate : STRING;
	YKoordinate : STRING;
	Theta : STRING;
	
	// Eingangsvariablen für die Funktion LREAL_TO_FMTSTR
	iPrecision : INT; // Definition Anzahl Nachkommastellen
	bRound     : BOOL; // String wird gerundet 
	
	sPayloadJobNumber : STRING(255);
	
	otherRobotNumbers : ARRAY[1..3] OF INT;
	
	// Flags, die zeigen, dass wir ein Topic bereits erfolgreich abonniert haben
	bSubscribedJobNumber : BOOL := FALSE;
	bSubscribedChargeConn1 : BOOL := FALSE;
	bSubscribedChargeConn2 : BOOL := FALSE;
	bSubscribedBumperReset : BOOL := FALSE;
	bSubscribedGlobalReset : BOOL := FALSE;
	bSubscribedPartLostReset : BOOL := FALSE;
	bSubscribedPosX : ARRAY[1..numRobots] OF BOOL := [numRobots(FALSE)];
	bSubscribedPosY : ARRAY[1..numRobots] OF BOOL := [numRobots(FALSE)];
	
	// Reset
	sTopicSubBumperReset : STRING(255);
	sTopicSubGlobalReset : STRING(255);
	sTopicSubPartLostReset : STRING(255);
	sPayloadBumperReset : STRING(255);
	sPayloadGlobalReset : STRING(255);
	sPayloadPartLostReset : STRING(255);
	
	bumperReset AT %Q* : BOOL := FALSE;
	globalReset AT %Q* : BOOL := FALSE;
	partLostReset AT %Q* : BOOL := FALSE;
	
	// Kommunikation mit Ladestation
	
	sTopicChargeConn1 : STRING(255) := ('Charging/Stat1');
	sPayloadChargeConn1: STRING (255);
	
	chargeConnect1: STRING (255);
	chargeStation1Connected AT %Q* : BOOL;
	chargeStation1Charging AT %Q* : BOOL;
	chargeStation1Completed AT %Q* : BOOL;
	
	sTopicChargeConn2 : STRING(255) := ('Charging/Stat2');
	sPayloadChargeConn2: STRING (255);
	
	chargeConnect2: STRING (255);
	chargeStation2Connected AT %Q* : BOOL;
	chargeStation2Charging AT %Q* : BOOL;
	chargeStation2Completed AT %Q* : BOOL;
	
	MyJob : STRING(255);  // Variable zur Speicherung der empfangenen Jobnummer
	myJobNum AT %Q* : INT := 0;
	
	// Akku Strom und Spannung
	supplyCurrent_A			AT%I* : REAL; 
	batteryVoltage_V		AT%I*  : REAL;
	sTopicPubToPowerMgmt : STRING(255);
	
	// Fehlermeldungen
	errorTextRobot AT %I*: STRING;

	iRobotNumber: INT;
	
	sTopicTemp: STRING(255);
	
	robotPositions AT %Q* : ARRAY[1..4] OF Position;
	x: INT;
	y: INT;
	e: INT;
	
	msgCounter : INT := 0;
	numMessagesDequeued : INT := 0;

	///////////////////////////MQTT GW4 //////////////////
	// Publish message
	initMQTT : BOOL := FALSE;

	sTopicPubToPowerMgmt_SOC : STRING(255);// := CONCAT('Robots/PowerMgmt/SoC_Robot_', INT_TO_STRING(.Var_HAWIno.Robot_Number)); 
	
	sTopicSubToPowerMgmt : STRING(255);// := CONCAT('PowerMgmt/Robots/Robot_', INT_TO_STRING(.Var_HAWIno.Robot_Number));
	hrErrorOccurred : HRESULT; 			// Enthlt dern letzten augetretenen Fehler
	
	// Variables for JSON
	fbJson			: FB_JsonSaxWriter;
	fbJsonDataType 	: FB_JsonReadWriteDataType;
	sJsonDoc       	: STRING(2000); 
	
	stMqtt_HAWino_IN	 AT%I*: ST_PwrMgmt_HAWino_In;		// Attention! Don't link TIME Variables, otherwise we get an error!
	stMqtt_HAWino_Out	 AT%Q*: ST_PwrMgmt_HAWino_Out;
	
	SOC_Out : STRING(255);
	nBatteryTemperature	AT%I*	: INT;
	
	bComCheckAnswer	AT%Q*	: BOOL;
	
	stMqtt_HAWinoValues	: ST_PwrMgmt_HAWino;
	
	// Timer to create a time stamp
	fbTimerTimestamp : TON := (PT:=T#71582M47S295MS);
	
	// Local Vaiables to evaluate and act to input
	fbComCheckFlag	: RS;
	
	
	sTopicSubToFleetMgmt: STRING;
	Reset1: BOOL;
	//Input synccheck. robotdata has been read and can be used.
	txtReadInit AT %I* : BOOL := FALSE;
	
	stMqtt_HAWino_I: INT;
	fActualBatteryVoltage: INT;
	FORMAT: INT;
	myValue: INT;
	value: INT;
	
	gewerk4pubcounter : INT := 0;
	
END_VAR

VAR CONSTANT
	sTopicPubCharge1 : STRING(255) := 'Charging/1/Load';
	sTopicPubCharge2 : STRING(255) := 'Charging/2/Load';
	
	numRobots: INT := 4;
END_VAR

IF bSetParameter THEN
	fbIotMqttClient.sHostName := IPAdress;	// IP-Adresse des Servers
	fbIotMqttClient.nHostPort := HostPort;
	//fbIotMqttClient.sClientId := ClientId;
	fbIotMqttClient.sClientId := CONCAT('Robot_', INT_TO_STRING(.Var_HAWIno.Robot_Number));
	fbIotMqttClient.sTopicPrefix := '';
	//fbIotMqttClient.nKeepAlive:= 60; 
	fbIotMqttClient.sUserName:= User;
	fbIotMqttClient.sUserPassword:= Password;
	//fbIotMqttClient.stWill:= ; 
	//fbIotMqttClient.stTLS:= ;
	fbIotMqttClient.ipMessageQueue := fbMessageQueue;

	bSetParameter := FALSE;
END_IF

fbIotMqttClient.Execute(bConnect);

////////////////////////////////////////////////////////////////////////////////////////////////////////////////////////////////////////////////////
/////////////////////////////////////////CHARGING-STATION do not delete///////////////////////////////////////////////
////////////////////////////////////////////////////////////////////////////////////////////////////////////////////////////////////////////////////


fbTimer(IN:=TRUE);

IF fbTimer.Q THEN // ALIVE BIT 
	fbTimer(IN:=FALSE);
	sPayloadPub := 'ALIVE';
	sTopicPubAlive := CONCAT('Robots/PowerMgmt/Robot_', INT_TO_STRING(.Var_HAWIno.Robot_Number));
	sTopicPubAlive := CONCAT (sTopicPubAlive, '/LifeBit');
	fbIotMqttClient.Publish(
		sTopic := sTopicPubAlive, 
		pPayload := ADR(sPayloadPub), nPayloadSize:= LEN2(ADR(sPayloadPub)), 
		eQoS := TcIotMqttQos.AtMostOnceDelivery, bRetain:= FALSE, bQueue:= FALSE
	);

END_IF	

// Neuer Timer für Batteriedaten außer SoC // Publish alle 5 Sekunden
fbTimerPubBat(IN:=TRUE);

IF fbTimerPubBat.Q THEN
	
	fbTimerPubBat(IN:=FALSE);
	
	sTopicPubToPowerMgmt := CONCAT('Robots/PowerMgmt/Robot_', INT_TO_STRING(.Var_HAWIno.Robot_Number));
	sTopicPubToPowerMgmt := CONCAT(sTopicPubToPowerMgmt, '/Voltage');
	//sPayloadPub:= REAL_TO_STRING(batteryVoltage_V); // 
	sPayloadPub := LREAL_TO_FMTSTR( batteryVoltage_V, 3, FALSE );
	fbIotMqttClient.Publish(sTopic:= sTopicPubToPowerMgmt, 
							pPayload:= ADR( sPayloadPub), 
							nPayloadSize:= LEN2(ADR( sPayloadPub)), 
							eQoS:= TcIotMqttQos.AtMostOnceDelivery, 
							bRetain:= FALSE, 
							bQueue:= FALSE);
							
	sTopicPubToPowerMgmt := CONCAT('Robots/PowerMgmt/Robot_', INT_TO_STRING(.Var_HAWIno.Robot_Number));
	sTopicPubToPowerMgmt := CONCAT(sTopicPubToPowerMgmt, '/Current');
	//sPayloadPub:= REAL_TO_STRING(supplyCurrent_A); // Der LREAL Wert soll auf zwei Stellen gerundet werden
	sPayloadPub := LREAL_TO_FMTSTR( supplyCurrent_A, 3, FALSE );
	fbIotMqttClient.Publish(sTopic:= sTopicPubToPowerMgmt, 
							pPayload:= ADR( sPayloadPub), 
							nPayloadSize:= LEN2(ADR( sPayloadPub)), 
							eQoS:= TcIotMqttQos.AtMostOnceDelivery, 
							bRetain:= FALSE, 
							bQueue:= FALSE);
							
							
	sTopicPubToPowerMgmt := CONCAT('Robots/PowerMgmt/Robot_', INT_TO_STRING(.Var_HAWIno.Robot_Number));
	sTopicPubToPowerMgmt := CONCAT(sTopicPubToPowerMgmt, '/Temperature');
	//sPayloadPub:= REAL_TO_STRING(supplyCurrent_A); // Der LREAL Wert soll auf zwei Stellen gerundet werden
	sPayloadPub := LREAL_TO_FMTSTR( stMqtt_HAWinoValues.Output.fBatteryTemperature, 3, TRUE );
	fbIotMqttClient.Publish(sTopic:= sTopicPubToPowerMgmt, 
							pPayload:= ADR( sPayloadPub), 
							nPayloadSize:= LEN2(ADR( sPayloadPub)), 
							eQoS:= TcIotMqttQos.AtMostOnceDelivery, 
							bRetain:= FALSE, 
							bQueue:= FALSE);
							
	sTopicPubToPowerMgmt := CONCAT('Robots/PowerMgmt/Robot_', INT_TO_STRING(.Var_HAWIno.Robot_Number));
	sTopicPubToPowerMgmt := CONCAT(sTopicPubToPowerMgmt, '/RunningTime');
	//sPayloadPub:= REAL_TO_STRING(supplyCurrent_A); // Der LREAL Wert soll auf zwei Stellen gerundet werden
	sPayloadPub := LREAL_TO_FMTSTR( stMqtt_HAWinoValues.Output.nEstimatedRunningTime, 0, TRUE );
	fbIotMqttClient.Publish(sTopic:= sTopicPubToPowerMgmt, 
							pPayload:= ADR( sPayloadPub), 
							nPayloadSize:= LEN2(ADR( sPayloadPub)), 
							eQoS:= TcIotMqttQos.AtMostOnceDelivery, 
							bRetain:= FALSE, 
							bQueue:= FALSE);
							
	sTopicPubToPowerMgmt := CONCAT('Robots/PowerMgmt/Robot_', INT_TO_STRING(.Var_HAWIno.Robot_Number));
	sTopicPubToPowerMgmt := CONCAT(sTopicPubToPowerMgmt, '/ChargingTime');
	sPayloadPub := LREAL_TO_FMTSTR( stMqtt_HAWinoValues.Output.nEstimatedChargingTime, 0, FALSE );
	fbIotMqttClient.Publish(sTopic:= sTopicPubToPowerMgmt, 
							pPayload:= ADR( sPayloadPub), 
							nPayloadSize:= LEN2(ADR( sPayloadPub)), 
							eQoS:= TcIotMqttQos.AtMostOnceDelivery, 
							bRetain:= FALSE, 
							bQueue:= FALSE);
							
	sTopicPubToPowerMgmt := CONCAT('Robots/PowerMgmt/Robot_', INT_TO_STRING(.Var_HAWIno.Robot_Number));
	sTopicPubToPowerMgmt := CONCAT(sTopicPubToPowerMgmt, '/CurrentDetected');
	sPayloadPub := BOOL_TO_STRING(supplyCurrent_A < 1.65 and supplyCurrent_A > 0);
	fbIotMqttClient.Publish(sTopic:= sTopicPubToPowerMgmt, 
							pPayload:= ADR( sPayloadPub), 
							nPayloadSize:= LEN2(ADR( sPayloadPub)), 
							eQoS:= TcIotMqttQos.AtMostOnceDelivery, 
							bRetain:= FALSE, 
							bQueue:= FALSE);
END_IF

fbTimerPubSoC(IN:=TRUE);
 // Publish SoC alle 10 Sekunden
 
IF fbTimerPubSoC.Q THEN
	
	fbTimerPubSoC(IN:=FALSE);
							
	sTopicPubToPowerMgmt := CONCAT('Robots/PowerMgmt/Robot_', INT_TO_STRING(.Var_HAWIno.Robot_Number));
	sTopicPubToPowerMgmt := CONCAT(sTopicPubToPowerMgmt, '/SoC');
	sPayloadPub := LREAL_TO_FMTSTR( stMqtt_HAWinoValues.Output.fSoC, 2, FALSE );
	fbIotMqttClient.Publish(sTopic:= sTopicPubToPowerMgmt, 
							pPayload:= ADR( sPayloadPub), 
							nPayloadSize:= LEN2(ADR( sPayloadPub)), 
							eQoS:= TcIotMqttQos.AtMostOnceDelivery, 
							bRetain:= FALSE, 
							bQueue:= FALSE);

END_IF





IF txtReadInit THEN
	IF NOT initMQTT THEN
		sTopicPubToPowerMgmt  := CONCAT('Robots/PowerMgmt/Robot_', INT_TO_STRING(.Var_HAWIno.Robot_Number));
		sTopicSubToPowerMgmt  := CONCAT('PowerMgmt/Robots/Robot_', INT_TO_STRING(.Var_HAWIno.Robot_Number));
		initMQTT:= TRUE;
	END_IF
	
	stMqtt_HAWinoValues.Output.nRobotNumber := .Var_HAWIno.Robot_Number;			// Anpassen für jeden HAWino
	
	fbTimerTimestamp(In:= NOT fbTimerTimestamp.Q, ET=>stMqtt_HAWinoValues.Output.tTimestamp);
	//SOC-Berechnung
	stMqtt_HAWinoValues.Output.fSoC := stMqtt_HAWino_In.fSoC; //Ausgabe direkt auf MQTT unter PowerMgmt->SoC_Robot_(no)

										
	stMqtt_HAWinoValues.Output.fActualBatteryCurrent := stMqtt_HAWino_In.fActualBatteryCurrent;
	stMqtt_HAWinoValues.Output.fActualBatteryVoltage := stMqtt_HAWino_In.fActualBatteryVoltage;

	// Skalierung der Temperaturwerte des Akkus
	stMqtt_HAWinoValues.Output.fBatteryTemperature := FKT_Scale(Rohwert := nBatteryTemperature, 
																	X1 := -500,
																	X2 := 1500, 
																	Y1 := -50,
																	Y2 := 150);
																	
	// Ausgabe der erwarteten Laufzeit des Roboters
	stMqtt_HAWinoValues.Output.nEstimatedRunningTime	:= LIMIT(0,stMqtt_HAWino_In.nEstimatedRunningTime,172800);		// Max. 48 Stunden sollen dargestellt werden
	stMqtt_HAWinoValues.Output.nEstimatedChargingTime	:= LIMIT(0,stMqtt_HAWino_In.nEstimatedChargingTime,172800);		// Max. 48 Stunden sollen dargestellt werden
		
	// Antworten auf den Kommunikationstest und des Ladetests
	stMqtt_HAWinoValues.Output.bCheckCurrentDetected := stMqtt_HAWino_In.bCheckCurrentDetected;
	stMqtt_HAWinoValues.Output.bComCheckAnswer := stMqtt_HAWino_In.bComCheckAnswer;

					
END_IF

END_PROGRAM

// ---- POUs/HAWinoCore/04_SystemManagment/FKT_Scale.TcPOU
FUNCTION FKT_Scale : LREAL
VAR_INPUT
	// Unterer Auflösungsbereich
	X1: LREAL;
	// Oberer Auflösungsbereich
	X2: LREAL;
	// Unterer Darstellungsbereich
	Y1: LREAL;
	// Oberer Darstellungsbereich
	Y2: LREAL;
END_VAR
VAR
	// Rohwert in Real
	X: LREAL;
	// Skalierter Messwert
	Y: LREAL := 0;
END_VAR
VAR_INPUT
	// Analoger Eingang in 12 bzw. 16 Bit
	Rohwert: LREAL;
END_VAR

X := Rohwert;

Y := ((((Y2-Y1)/(X2-X1))*(X-X1))+Y1);			// Skalierung über eine lineare Funktion

IF Y > Y2 THEN
	Y := Y2;									// Obere Begrenzung
ELSIF Y < Y1 THEN
	Y := Y1;									// Untere Begrenzung
END_IF

FKT_Scale := Y;									// Ausgabe

END_FUNCTION

// ---- POUs/HAWinoCore/02_IR-Sensors/IrDistanceSensors.TcPOU
PROGRAM IrDistanceSensors
VAR
	distanceRaw AT %I* : ARRAY [1..9] OF INT;
	
	distance_mm AT %Q* : ARRAY [1..9] OF LREAL;

	i : INT;
END_VAR

FOR  i := 1 TO 9 DO
	distance_mm[i] := IrDistanceFromRaw(distanceRaw[i]);
END_FOR

END_PROGRAM

// ---- POUs/HAWinoCore/02_IR-Sensors/IrDistanceFromRaw.TcPOU
FUNCTION IrDistanceFromRaw : LREAL
VAR_INPUT
	rawValue : INT;
END_VAR
VAR
END_VAR

	IrDistanceFromRaw := 123.15 / EXPT( INT_TO_REAL(rawValue) * (10.0 / 32767.0), 1.119 );

END_FUNCTION

// ---- POUs/HAWinoCore/03_Communication/Camera.TcPOU
PROGRAM Camera
VAR
		cameraData : CameraConnectionUDP;
END_VAR

cameraData();

END_PROGRAM

// ---- POUs/HAWinoCore/03_Communication/CameraConnectionUDP.TcPOU
{attribute 'c++_compatible'}
FUNCTION_BLOCK CameraConnectionUDP IMPLEMENTS ITcIoUdpProtocolRecv
VAR_INPUT
END_VAR
VAR_OUTPUT
	robotPosition AT %Q* : ARRAY [1..8] OF Position; 
	
	HH					AT	%Q*	:	LREAL;	
	MM					AT	%Q*	:	LREAL;
	SS					AT	%Q*	:	LREAL;
	MS					AT	%Q*	:	LREAL;
END_VAR
VAR
	{attribute 'TcInitSymbol'}
	oid : OTCID; // To be set in PLC_Instance object and required for FW_ObjMgr_GetObjectInstance()
	ipUdp : ITcIoUdpProtocol;
	nUdpPort : UINT := 25000;
	nReceivedPakets : UINT;
	//uLastReceivedIP : U_IpAdr; 
	hrInit : HRESULT;
	hrSend  : HRESULT; 	
	counter	:	UDINT	:= 0;
END_VAR


IF ipUdp <> 0 THEN
	ipUdp.CheckReceived();
END_IF

{attribute 'conditionalshow'}
METHOD FB_exit : BOOL
VAR_INPUT
	bInCopyCode : BOOL; // if TRUE, the exit method is called for exiting an instance that is copied afterwards (online change).
END_VAR
IF NOT bInCopyCode THEN // no online change
	IF ipUdp <> 0 THEN 
		ipUdp.UnregisterReceiver(nUdpPort); // Shutdown
		FW_SafeRelease(ADR(ipUdp));
		FB_exit := TRUE; 
	END_IF
END_IF
END_METHOD

{attribute 'conditionalshow'}
METHOD FB_init : BOOL
VAR_INPUT
	bInitRetains : BOOL; // if TRUE, the retain variables are initialized (warm start / cold start)
	bInCopyCode : BOOL;  // if TRUE, the instance afterwards gets moved into the copy code (online change)
END_VAR
VAR
	ipSrv : ITComObjectServer;
END_VAR
IF NOT bInCopyCode THEN // no online change
	IF ipUdp = 0 THEN
	    hrInit := FW_ObjMgr_GetObjectInstance(	oid:=oid, 
											iid:=TC_GLOBAL_IID_LIST.IID_ITcIoUdpProtocol, 
											pipUnk:=ADR(ipUdp) );
		IF SUCCEEDED(hrInit) THEN 
			IF  SUCCEEDED(ipUdp.RegisterReceiver(nUdpPort, THIS^)) THEN //open port
				FB_init := TRUE;
			ELSE 
				FW_SafeRelease(ADR(ipUdp));
			END_IF
		END_IF				
	END_IF
END_IF
END_METHOD

{attribute 'conditionalshow'}
METHOD FB_reinit : BOOL
VAR_INPUT
END_VAR
IF (ipUdp <> 0) THEN 
	ipUdp.RegisterReceiver(nUdpPort, THIS^);
	FB_reinit := TRUE; 
END_IF
END_METHOD

{attribute 'object_name' := 'ReceiveData'}
{attribute 'c++_compatible'}
{attribute 'signature_flag' := '33554688'}
{attribute 'pack_mode' := '4'}
{attribute 'show'}
{attribute 'minimal_input_size' := '4'}
METHOD ReceiveData : HRESULT
VAR_INPUT
	ipAddr	: UDINT;
	udpDestPort	: UINT;
	udpSrcPort	: UINT;
	nData	: UDINT;
	pData	: PVOID;
	pVlan	: POINTER TO ETYPE_VLAN_HEADER := 0;
END_VAR
VAR 
	i : INT;
	x,y,theta,e : LREAL;
	
END_VAR
nReceivedPakets := nReceivedPakets+1;
//uLastReceivedIP.ipAdrInternal := ipAddr;


	(*** Auslesen des Datenbereichs von UDP-Paketen ***
	* UDP-Telegramm besteht aus 56*8 = 448 Bytes (siehe UDP-Doku Lokalisierungsrechner)
	  Pro Robotino: 4*8 = 32 Bytes: je 8 Bytes für x-Koord, y-Koord, theta in rad, e
	  Robotino1: Bytes 1-8   -> x-Koord, Bytes 9-16  -> y-Koord, Bytes 17-24 -> theta
	  Robotino2: Bytes 25-32 -> x-Koord, Bytes 33-40 -> y-Koord, Bytes 41-48 -> theta  usw.. 
	* pData zeigt auf Adressbereich, in dem die 448 Byte großen UDP-Daten liegen
	  in der Schleife werden jeweils 8 Byte in den UDP-Array geschrieben und der Pointer nach
	  jedem Schritt um 8 Byte weiter geschoben.*)
	
IF nData = 448 THEN

	FOR i := 1 TO 8 DO
		memcpy( ADR(x), 	pData + 8 * 0 + 4*8*(i-1), 8);			// x-Koord
		memcpy( ADR(y),    	pData + 8 * 1 + 4*8*(i-1), 8);			// y-Koord
		memcpy( ADR(theta), pData + 8 * 2 + 4*8*(i-1), 8);			// theta
		memcpy( ADR(e), 	pData + 8 * 3 + 4*8*(i-1), 8);			// e
		
		robotPosition[i].x  := (x);
		robotPosition[i].y := (y);
		robotPosition[i].theta := (theta);
		robotPosition[i].e := (e);
			
	END_FOR
	
	memcpy( ADR(HH), pData + 256, 8);						// Hours
	memcpy( ADR(MM), pData + 264, 8);						// Minutes
	memcpy( ADR(SS), pData + 272, 8);						// Seconds
	memcpy( ADR(MS), pData + 280, 8);						// Milliseconds
END_IF
END_METHOD

{attribute 'object_name' := 'TcAddRef'}
{attribute 'c++_compatible'}
{attribute 'signature_flag' := '33554688'}
{attribute 'pack_mode' := '4'}
{attribute 'show'}
{attribute 'minimal_input_size' := '4'}
METHOD TcAddRef : UDINT
END_METHOD

{attribute 'object_name' := 'TcQueryInterface'}
{attribute 'c++_compatible'}
{attribute 'signature_flag' := '33554688'}
{attribute 'pack_mode' := '4'}
{attribute 'show'}
{attribute 'minimal_input_size' := '4'}
METHOD TcQueryInterface : HRESULT
VAR_INPUT
	iid	: REFERENCE TO IID;
	pipItf	: POINTER TO PVOID;
END_VAR
VAR
	ipUdpRecv : ITcIoUdpProtocolRecv;
	ipUnknown : ITcUnknown;	
END_VAR
IF GuidsEqual(ADR(iid), ADR(TC_GLOBAL_IID_LIST.IID_ITcIoUdpProtocolRecv)) THEN
	ipUdpRecv := THIS^; // cast to interface pointer
	pipItf^ := ITCUNKNOWN_TO_PVOID(ipUdpRecv);
	TcAddRef();
	TcQueryInterface := S_OK;
ELSIF GuidsEqual(ADR(iid), ADR(TC_GLOBAL_IID_LIST.IID_ITcUnknown)) THEN
	ipUnknown := THIS^; // cast to interface pointer
	pipItf^ := ITCUNKNOWN_TO_PVOID(ipUnknown);
	TcAddRef();
	TcQueryInterface := S_OK;
ELSE
	TcQueryInterface := E_HRESULTAdsErr.NOINTERFACE ; //Call super if this fb extends some other
END_IF
END_METHOD

{attribute 'object_name' := 'TcRelease'}
{attribute 'c++_compatible'}
{attribute 'signature_flag' := '33554688'}
{attribute 'pack_mode' := '4'}
{attribute 'show'}
{attribute 'minimal_input_size' := '4'}
METHOD TcRelease : UDINT
END_METHOD

END_FUNCTION_BLOCK

// ---- POUs/HAWinoCore/05_Bahnplanung/FB_MQTTNeu.TcPOU
FUNCTION_BLOCK FB_MQTTNeu
VAR
    fbClient            : FB_IotMqttClient;
    fbMessageQueue      : FB_IotMqttMessageQueue;
    fbMessage           : FB_IotMqttMessage;
    bSubscribed         : BOOL;
    sReceived           : STRING;

    bSendError          : BOOL;
    bSendJob            : BOOL;
    bSendState          : BOOL;
    bSendToken          : BOOL;

    sReceivedjob        : STRING(1000);
    sReceivedcmd        : STRING(1000);
    sReceivedStart      : STRING;
    sReceivedToken      : STRING;
	sReceivedChargingStatus : STRING;

    sSendError          : STRING(1000);
    sSendJob            : STRING(1000);
    sSendState          : STRING(1000);
    sSendToken          : STRING(1000);
    sSendCharging       : STRING;
    sSendStop           : STRING;

    sMqttSEND           : sMqttOut;
    sMqttRECEIVE        : sMqttIn;

    // JSON Parser
    fbJson              : FB_JsonDomParser;
    jsonDoc             : SJsonValue;
    jsonNode            : SJsonValue;

    // Topics (Subscribe)
    tempjob             : STRING;
    tempcmd             : STRING;
    tempInit            : STRING;
    temprToken          : STRING;

    // Topics (Publish)
    tempserror          : STRING;
    tempsjob            : STRING;
    tempsstate          : STRING;
    tempstoken          : STRING;

    // Hilfsvariablen
    start               : BOOL;
    LADEN               : BOOL;
    charging_dock       : INT;
    loading_speed       : INT;
    station_id          : STRING;
    TONPosition         : TON;
    boTONFlanke         : BOOL;
	sReceivedPoint1		: STRING;
	sReceivedPoint2		: STRING;
	incharging_point1	: INT;
	incharging_point2	: INT;
	Charging			: BOOL;
	

    // Flags: neue Nachricht auf Topic eingegangen
    bNewMsgCmd          : BOOL;
    bNewMsgJob          : BOOL;
    bNewMsgToken        : BOOL;

    // Change-Detection Senden: Error-Topic
    prevErrorRoutePlanning  : BOOL;
    prevErrorControl        : BOOL;
    prevErrorNoWorkpiece    : BOOL;
    prevErrorWorkpieceLost  : BOOL;

    // Change-Detection Senden: JobState-Topic
    prevWorkpieceLoaded     : BOOL;
    prevTransportWorkpiece  : BOOL;
    prevJobAccepted         : BOOL;
    prevWaitForRfidOut      : BOOL;
    prevWaitForRfidIn       : BOOL;
    prevWorkpiecePlaced     : BOOL;

    // Change-Detection Senden: Token-Topic
    prevTokenRequest        : BOOL;
    prevTokenRelease        : BOOL;

END_VAR
VAR_INPUT
    xsDataToSend            : sMqttOut;
    xsKoordinate            : sKoordinate;
    xinMqttTokenTargetId    : INT;
	xboCharging				: BOOL;
	xinChargingPoint		: INT;
END_VAR
VAR_OUTPUT
    ysDataToReceive         : sMqttIn;
	yinchargingstatus		: INT;
END_VAR

// ============================================================
// Verbindungsparameter
// ============================================================
fbClient.sHostName      := '192.168.0.11';
fbClient.nHostPort      := 1883;
fbClient.sUserName      := 'VPJ';
fbClient.sUserPassword  := 'R462';


CASE Robot_Number OF 
	1: fbClient.sClientId := 'Eis1';
	2: fbClient.sClientId := 'Eis2';
	3: fbClient.sClientId := 'Eis3';
	4: fbClient.sClientId := 'Eis4';
END_CASE





fbClient.ipMessageQueue := fbMessageQueue;
fbClient.Execute(bConnect := TRUE);

sMqttSEND := xsDataToSend;

// ============================================================
// Alle empfangenen Bools zu Beginn jedes Zyklus zuruecksetzen.
// Sie sind nur TRUE wenn in diesem Zyklus eine neue Nachricht kam.
// ============================================================
sMqttRECEIVE.sCmd.boStop            := FALSE;
sMqttRECEIVE.sCmd.boReset           := FALSE;
sMqttRECEIVE.sCmd.boJobReset        := FALSE;
sMqttRECEIVE.sCmd.boRFIDComplete    := FALSE;
sMqttRECEIVE.sCmd.boStartJob        := FALSE;
sMqttRECEIVE.sCmd.boTokenGrant      := FALSE;
sMqttRECEIVE.sCmd.boCancelCharging  := FALSE;
bNewMsgCmd                          := FALSE;
bNewMsgJob                          := FALSE;
bNewMsgToken                        := FALSE;
sMqttRECEIVE.boNewJob := FALSE;

// ============================================================
// Einmalig subscriben wenn verbunden
// ============================================================
IF fbClient.bConnected AND NOT bSubscribed THEN

    tempjob := CONCAT('HAWino/', INT_TO_STRING(Robot_Number));
    tempjob := CONCAT(tempjob, '/job');
    fbClient.Subscribe(sTopic := tempjob, eQoS := 0);

    tempcmd := CONCAT('HAWino/', INT_TO_STRING(Robot_Number));
    tempcmd := CONCAT(tempcmd, '/cmd');
    fbClient.Subscribe(sTopic := tempcmd, eQoS := 0);

    tempInit := CONCAT('HAWino/', INT_TO_STRING(Robot_Number));
    tempInit := CONCAT(tempInit, '/init');
    fbClient.Subscribe(sTopic := tempInit, eQoS := 0);

    temprToken := CONCAT('HAWino/', INT_TO_STRING(Robot_Number));
    temprToken := CONCAT(temprToken, '/token');
    fbClient.Subscribe(sTopic := temprToken, eQoS := 0);
	
	fbClient.Subscribe(sTopic := 'ChargingPointStatus/+', eQoS := 0);
	
	fbClient.Subscribe(sTopic := 'ChargingStatus/+', eQoS := 0);

    tempserror := CONCAT('HAWino/', INT_TO_STRING(Robot_Number));
    tempserror := CONCAT(tempserror, '/error');

    tempsjob := CONCAT('HAWino/', INT_TO_STRING(Robot_Number));
    tempsjob := CONCAT(tempsjob, '/jobState');

    tempsstate := CONCAT('HAWino/', INT_TO_STRING(Robot_Number));
    tempsstate := CONCAT(tempsstate, '/generalState');

    bSubscribed := TRUE;
END_IF

// ============================================================
// Nachrichten aus Queue lesen
// ============================================================
IF fbMessageQueue.nQueuedMessages > 0 THEN

    fbMessageQueue.Dequeue(fbMessage := fbMessage);
    fbMessage.GetPayload(
        pPayload            := ADR(sReceived),
        nPayloadSize        := SIZEOF(sReceived),
        bSetNullTermination := TRUE
    );

    IF fbMessage.CompareTopic(sTopic := tempjob) THEN
        fbMessage.GetPayload(pPayload := ADR(sReceivedjob),   nPayloadSize := SIZEOF(sReceivedjob),   bSetNullTermination := TRUE);
        bNewMsgJob := TRUE;
		sMqttRECEIVE.boNewJob := TRUE;
    ELSIF fbMessage.CompareTopic(sTopic := tempcmd) THEN
        fbMessage.GetPayload(pPayload := ADR(sReceivedcmd),   nPayloadSize := SIZEOF(sReceivedcmd),   bSetNullTermination := TRUE);
        bNewMsgCmd := TRUE;
    ELSIF fbMessage.CompareTopic(sTopic := tempInit) THEN
        fbMessage.GetPayload(pPayload := ADR(sReceivedStart), nPayloadSize := SIZEOF(sReceivedStart), bSetNullTermination := TRUE);
    ELSIF fbMessage.CompareTopic(sTopic := temprToken) THEN
        fbMessage.GetPayload(pPayload := ADR(sReceivedToken), nPayloadSize := SIZEOF(sReceivedToken), bSetNullTermination := TRUE);
        bNewMsgToken := TRUE;
	ELSIF fbMessage.CompareTopic(sTopic := 'ChargingPointStatus/Point1') THEN
        fbMessage.GetPayload(pPayload := ADR(sReceivedPoint1), nPayloadSize := SIZEOF(sReceivedPoint1), bSetNullTermination := TRUE);
        bNewMsgToken := TRUE;
	ELSIF fbMessage.CompareTopic(sTopic := 'ChargingPointStatus/Point2') THEN
        fbMessage.GetPayload(pPayload := ADR(sReceivedPoint2), nPayloadSize := SIZEOF(sReceivedPoint2), bSetNullTermination := TRUE);
        bNewMsgToken := TRUE;
	ELSIF fbMessage.CompareTopic(sTopic := 'ChargingStatus') THEN
        fbMessage.GetPayload(pPayload := ADR(sReceivedChargingStatus), nPayloadSize := SIZEOF(sReceivedChargingStatus), bSetNullTermination := TRUE);
        bNewMsgToken := TRUE;
    END_IF

END_IF

// ============================================================
// JSON parsen: CMD (nur wenn neue Nachricht)
// ============================================================
IF bNewMsgCmd THEN
    jsonDoc := fbJson.ParseDocument(sReceivedcmd);
    IF jsonDoc <> 0 THEN

        jsonNode := fbJson.FindMember(jsonDoc, 'boStop');
        IF jsonNode <> 0 THEN
            sMqttRECEIVE.sCmd.boStop := fbJson.GetBool(jsonNode);
        END_IF

        jsonNode := fbJson.FindMember(jsonDoc, 'boReset');
        IF jsonNode <> 0 THEN
            sMqttRECEIVE.sCmd.boReset := fbJson.GetBool(jsonNode);
        END_IF

        jsonNode := fbJson.FindMember(jsonDoc, 'boJobReset');
        IF jsonNode <> 0 THEN
            sMqttRECEIVE.sCmd.boJobReset := fbJson.GetBool(jsonNode);
        END_IF

        jsonNode := fbJson.FindMember(jsonDoc, 'boRfidComplete');
        IF jsonNode <> 0 THEN
            sMqttRECEIVE.sCmd.boRFIDComplete := fbJson.GetBool(jsonNode);
        END_IF

        jsonNode := fbJson.FindMember(jsonDoc, 'boStartJob');
        IF jsonNode <> 0 THEN
            sMqttRECEIVE.sCmd.boStartJob := fbJson.GetBool(jsonNode);
        END_IF

        jsonNode := fbJson.FindMember(jsonDoc, 'boCancelCharging');
        IF jsonNode <> 0 THEN
            sMqttRECEIVE.sCmd.boCancelCharging := fbJson.GetBool(jsonNode);
        END_IF

    END_IF
    // String leeren damit kein alter Inhalt im naechsten Zyklus nochmal geparsed wird
    sReceivedcmd := '';
END_IF

// ============================================================
// JSON parsen: JOB (nur wenn neue Nachricht)
// Hinweis: JobID/Destinations sind keine Einzel-Pulse, die bleiben
// als letzter empfangener Wert erhalten (kein Reset noetig)
// ============================================================
IF bNewMsgJob THEN
    jsonDoc := fbJson.ParseDocument(sReceivedjob);
    IF jsonDoc <> 0 THEN

        jsonNode := fbJson.FindMember(jsonDoc, 'jobId');
        IF jsonNode <> 0 THEN
            sMqttRECEIVE.sJOB.inJobID := DINT_TO_INT(fbJson.GetInt(jsonNode));
        END_IF

        jsonNode := fbJson.FindMember(jsonDoc, 'inDestination1');
        IF jsonNode <> 0 THEN
            sMqttRECEIVE.sJOB.inDestination1 := DINT_TO_INT(fbJson.GetInt(jsonNode));
        END_IF

        jsonNode := fbJson.FindMember(jsonDoc, 'inDestination2');
        IF jsonNode <> 0 THEN
            sMqttRECEIVE.sJOB.inDestination2 := DINT_TO_INT(fbJson.GetInt(jsonNode));
        END_IF

    END_IF
    sReceivedjob := '';
END_IF

// ============================================================
// JSON parsen: TOKEN (nur wenn neue Nachricht)
// ============================================================
IF bNewMsgToken THEN
    jsonDoc := fbJson.ParseDocument(sReceivedToken);
    IF jsonDoc <> 0 THEN
        jsonNode := fbJson.FindMember(jsonDoc, 'category');
        IF jsonNode <> 0 THEN
            IF fbJson.GetString(jsonNode) = 'TOKEN_GRANT' THEN
                sMqttRECEIVE.sCmd.boTokenGrant := TRUE;
            END_IF
        END_IF
    END_IF
    // String leeren damit boTokenGrant im naechsten Zyklus wieder FALSE ist
    sReceivedToken := '';
END_IF

//State of Charging auslesen
jsonDoc := fbJson.ParseDocument(sReceivedChargingStatus);
   IF jsonDoc <> 0 THEN

       jsonNode := fbJson.FindMember(jsonDoc, 'state_of_charging');
       IF jsonNode <> 0 THEN
            yinchargingstatus := DINT_TO_INT(fbJson.GetInt(jsonNode));
       END_IF
	END_IF

// ============================================================
// Senden
// ============================================================
start := TRUE;

IF start THEN

    // ----------------------------------------------------------
    // ERROR TOPIC: nur geaenderte Bools einzeln senden
    // ----------------------------------------------------------
    IF sMqttSEND.sError.boErrorRoutePlanning <> prevErrorRoutePlanning THEN
        prevErrorRoutePlanning := sMqttSEND.sError.boErrorRoutePlanning;
        IF fbClient.bConnected THEN
            IF sMqttSEND.sError.boErrorRoutePlanning THEN
                sSendError := '{"boErrorRoutePlanning":true}';
            ELSE
                sSendError := '{"boErrorRoutePlanning":false}';
            END_IF
            fbClient.Publish(
                sTopic       := tempserror,
                pPayload     := ADR(sSendError),
                nPayloadSize := LEN(sSendError),
                eQoS         := 0,
                bRetain      := FALSE,
                bQueue       := FALSE
            );
        END_IF
    END_IF

    IF sMqttSEND.sError.boErrorControl <> prevErrorControl THEN
        prevErrorControl := sMqttSEND.sError.boErrorControl;
        IF fbClient.bConnected THEN
            IF sMqttSEND.sError.boErrorControl THEN
                sSendError := '{"boErrorControl":true}';
            ELSE
                sSendError := '{"boErrorControl":false}';
            END_IF
            fbClient.Publish(
                sTopic       := tempserror,
                pPayload     := ADR(sSendError),
                nPayloadSize := LEN(sSendError),
                eQoS         := 0,
                bRetain      := FALSE,
                bQueue       := FALSE
            );
        END_IF
    END_IF

    IF sMqttSEND.sError.boErrorNoWorkpiece <> prevErrorNoWorkpiece THEN
        prevErrorNoWorkpiece := sMqttSEND.sError.boErrorNoWorkpiece;
        IF fbClient.bConnected THEN
            IF sMqttSEND.sError.boErrorNoWorkpiece THEN
                sSendError := '{"boErrorNoWorkpiece":true}';
            ELSE
                sSendError := '{"boErrorNoWorkpiece":false}';
            END_IF
            fbClient.Publish(
                sTopic       := tempserror,
                pPayload     := ADR(sSendError),
                nPayloadSize := LEN(sSendError),
                eQoS         := 0,
                bRetain      := FALSE,
                bQueue       := FALSE
            );
        END_IF
    END_IF

    IF sMqttSEND.sError.boErrorWorkpieceLost <> prevErrorWorkpieceLost THEN
        prevErrorWorkpieceLost := sMqttSEND.sError.boErrorWorkpieceLost;
        IF fbClient.bConnected THEN
            IF sMqttSEND.sError.boErrorWorkpieceLost THEN
                sSendError := '{"boErrorWorkpieceLost":true}';
            ELSE
                sSendError := '{"boErrorWorkpieceLost":false}';
            END_IF
            fbClient.Publish(
                sTopic       := tempserror,
                pPayload     := ADR(sSendError),
                nPayloadSize := LEN(sSendError),
                eQoS         := 0,
                bRetain      := FALSE,
                bQueue       := FALSE
            );
        END_IF
    END_IF

    // ----------------------------------------------------------
    // JOBSTATE TOPIC: nur geaenderte Bools einzeln senden
    // ----------------------------------------------------------
    IF sMqttSEND.sJobState.boWorkpieceLoaded <> prevWorkpieceLoaded THEN
        prevWorkpieceLoaded := sMqttSEND.sJobState.boWorkpieceLoaded;
        IF fbClient.bConnected THEN
            IF sMqttSEND.sJobState.boWorkpieceLoaded THEN
                sSendJob := '{"boWorkpieceLoaded":true}';
            ELSE
                sSendJob := '{"boWorkpieceLoaded":false}';
            END_IF
            fbClient.Publish(
                sTopic       := tempsjob,
                pPayload     := ADR(sSendJob),
                nPayloadSize := LEN(sSendJob),
                eQoS         := 0,
                bRetain      := FALSE,
                bQueue       := FALSE
            );
        END_IF
    END_IF

    IF sMqttSEND.sJobState.boTransportWorkpiece <> prevTransportWorkpiece THEN
        prevTransportWorkpiece := sMqttSEND.sJobState.boTransportWorkpiece;
        IF fbClient.bConnected THEN
            IF sMqttSEND.sJobState.boTransportWorkpiece THEN
                sSendJob := '{"boTransportWorkpiece":true}';
            ELSE
                sSendJob := '{"boTransportWorkpiece":false}';
            END_IF
            fbClient.Publish(
                sTopic       := tempsjob,
                pPayload     := ADR(sSendJob),
                nPayloadSize := LEN(sSendJob),
                eQoS         := 0,
                bRetain      := FALSE,
                bQueue       := FALSE
            );
        END_IF
    END_IF

    IF sMqttSEND.sJobState.boJobAccepted <> prevJobAccepted THEN
        prevJobAccepted := sMqttSEND.sJobState.boJobAccepted;
        IF fbClient.bConnected THEN
            IF sMqttSEND.sJobState.boJobAccepted THEN
                sSendJob := '{"boJobAccepted":true}';
            ELSE
                sSendJob := '{"boJobAccepted":false}';
            END_IF
            fbClient.Publish(
                sTopic       := tempsjob,
                pPayload     := ADR(sSendJob),
                nPayloadSize := LEN(sSendJob),
                eQoS         := 0,
                bRetain      := FALSE,
                bQueue       := FALSE
            );
        END_IF
    END_IF

    IF sMqttSEND.sJobState.boWaitForRfidOut <> prevWaitForRfidOut THEN
        prevWaitForRfidOut := sMqttSEND.sJobState.boWaitForRfidOut;
        IF fbClient.bConnected THEN
            IF sMqttSEND.sJobState.boWaitForRfidOut THEN
                sSendJob := '{"boWaitForRfidOut":true}';
            ELSE
                sSendJob := '{"boWaitForRfidOut":false}';
            END_IF
            fbClient.Publish(
                sTopic       := tempsjob,
                pPayload     := ADR(sSendJob),
                nPayloadSize := LEN(sSendJob),
                eQoS         := 0,
                bRetain      := FALSE,
                bQueue       := FALSE
            );
        END_IF
    END_IF

    IF sMqttSEND.sJobState.boWaitForRfidIn <> prevWaitForRfidIn THEN
        prevWaitForRfidIn := sMqttSEND.sJobState.boWaitForRfidIn;
        IF fbClient.bConnected THEN
            IF sMqttSEND.sJobState.boWaitForRfidIn THEN
                sSendJob := '{"boWaitForRfidIn":true}';
            ELSE
                sSendJob := '{"boWaitForRfidIn":false}';
            END_IF
            fbClient.Publish(
                sTopic       := tempsjob,
                pPayload     := ADR(sSendJob),
                nPayloadSize := LEN(sSendJob),
                eQoS         := 0,
                bRetain      := FALSE,
                bQueue       := FALSE
            );
        END_IF
    END_IF

    IF sMqttSEND.sJobState.boWorkpiecePlaced <> prevWorkpiecePlaced THEN
        prevWorkpiecePlaced := sMqttSEND.sJobState.boWorkpiecePlaced;
        IF fbClient.bConnected THEN
            IF sMqttSEND.sJobState.boWorkpiecePlaced THEN
                sSendJob := '{"boWorkpiecePlaced":true}';
            ELSE
                sSendJob := '{"boWorkpiecePlaced":false}';
            END_IF
            fbClient.Publish(
                sTopic       := tempsjob,
                pPayload     := ADR(sSendJob),
                nPayloadSize := LEN(sSendJob),
                eQoS         := 0,
                bRetain      := FALSE,
                bQueue       := FALSE
            );
        END_IF
    END_IF

    // ----------------------------------------------------------
    // GENERALSTATE TOPIC: periodisch senden (unveraendert)
    // ----------------------------------------------------------
    sMqttSEND.sGeneralState.strPosition := CONCAT(
        CONCAT(REAL_TO_STRING(xsKoordinate.rePosX), ','),
        REAL_TO_STRING(xsKoordinate.rePosY)
    );

    IF sMqttSEND.sGeneralState.boReady THEN
        sSendState := '{"boReady":true,"boCharging":';
    ELSE
        sSendState := '{"boReady":false,"boCharging":';
    END_IF
    IF sMqttSEND.sGeneralState.boCharging THEN
        sSendState := CONCAT(sSendState, 'true,"strPosition":"');
    ELSE
        sSendState := CONCAT(sSendState, 'false,"strPosition":"');
    END_IF
    sSendState := CONCAT(sSendState, sMqttSEND.sGeneralState.strPosition);
    sSendState := CONCAT(sSendState, '"}');

    TONPosition(IN := NOT boTONFlanke, PT := T#0.1S);
    boTONFlanke := TONPosition.Q;

    IF boTONFlanke AND fbClient.bConnected THEN
        fbClient.Publish(
            sTopic       := tempsstate,
            pPayload     := ADR(sSendState),
            nPayloadSize := LEN(sSendState),
            eQoS         := 0,
            bRetain      := FALSE,
            bQueue       := FALSE
        );
    END_IF

    // ----------------------------------------------------------
    // TOKEN TOPIC: nur bei Flanke senden
    // ----------------------------------------------------------
    CASE xinMqttTokenTargetId OF
        1: station_id := 'storage_1';
        2: station_id := 'storage_2';
        3: station_id := 'manufacturing_1';
        4: station_id := 'manufacturing_2';
        5: station_id := 'manufacturing_3';
		6: station_id := 'manufacturing_4';
		7: station_id := 'manufacturing_5';
		8: station_id := 'dispatch';
    END_CASE
    tempstoken := CONCAT('agents/station/', station_id);
    tempstoken := CONCAT(tempstoken, '/token');

    IF sMqttSEND.sToken.boTokenRequest <> prevTokenRequest THEN
        prevTokenRequest := sMqttSEND.sToken.boTokenRequest;
        IF sMqttSEND.sToken.boTokenRequest AND fbClient.bConnected THEN
            sSendToken := CONCAT('{"category":"TOKEN_REQUEST","robot_id":', INT_TO_STRING(Robot_Number));
            sSendToken := CONCAT(sSendToken, '}');
            fbClient.Publish(
                sTopic       := tempstoken,
                pPayload     := ADR(sSendToken),
                nPayloadSize := LEN(sSendToken),
                eQoS         := 0,
                bRetain      := FALSE,
                bQueue       := FALSE
            );
        END_IF
    END_IF

    IF sMqttSEND.sToken.boTokenRelease <> prevTokenRelease THEN
        prevTokenRelease := sMqttSEND.sToken.boTokenRelease;
        IF sMqttSEND.sToken.boTokenRelease AND fbClient.bConnected THEN
            sSendToken := CONCAT('{"category":"TOKEN_RELEASE","robot_id":', INT_TO_STRING(Robot_Number));
            sSendToken := CONCAT(sSendToken, '}');
            fbClient.Publish(
                sTopic       := tempstoken,
                pPayload     := ADR(sSendToken),
                nPayloadSize := LEN(sSendToken),
                eQoS         := 0,
                bRetain      := FALSE,
                bQueue       := FALSE
            );
        END_IF
    END_IF
	
	//Ladevorgang starten
	incharging_point1 := STRING_TO_INT(sReceivedPoint1);
	incharging_point2 := STRING_TO_INT(sReceivedPoint2);
	IF incharging_point1 = 1 THEN
		sMqttRECEIVE.boCharging1Connected := TRUE;
	ELSE
		sMqttRECEIVE.boCharging1Connected := FALSE;
	END_IF
	IF incharging_point2 = 1 THEN
		sMqttRECEIVE.boCharging2Connected := TRUE;
	ELSE
		sMqttRECEIVE.boCharging2Connected := FALSE;
	END_IF
	IF xboCharging AND fbClient.bConnected AND incharging_point1 = 1 AND (xinChargingPoint = 1) AND NOT Charging THEN
		sSendCharging := CONCAT('{"robot":', INT_TO_STRING(Robot_Number));
		sSendCharging := CONCAT(sSendCharging, ',"charge":true,"charging_dock":1,"loading_speed":100}');
	    fbClient.Publish(
            sTopic       := 'ChargingRequest',
            pPayload     := ADR(sSendCharging),
            nPayloadSize := LEN(sSendCharging),
            eQoS         := 0,
            bRetain      := FALSE,
            bQueue       := FALSE
         );
		 Charging := TRUE;
	END_IF
	
	IF xboCharging AND fbClient.bConnected AND incharging_point2 = 1 AND (xinChargingPoint = 2) AND NOT Charging THEN
		sSendCharging := CONCAT('{"robot":', INT_TO_STRING(Robot_Number));
		sSendCharging := CONCAT(sSendCharging, ',"charge":true,"charging_dock":2,"loading_speed":100}');
		fbClient.Publish(
            sTopic       := 'ChargingRequest',
            pPayload     := ADR(sSendCharging),
            nPayloadSize := LEN(sSendCharging),
            eQoS         := 0,
            bRetain      := FALSE,
            bQueue       := FALSE
         );
		 Charging := TRUE;
	END_IF
	
	IF (sMqttRECEIVE.sCmd.boCancelCharging OR sMqttRECEIVE.sCmd.boJobReset) AND fbClient.bConnected AND incharging_point1 = 1 AND (xinChargingPoint = 1) AND Charging THEN
		sSendCharging := CONCAT('{"robot":', INT_TO_STRING(Robot_Number));
		sSendCharging := CONCAT(sSendCharging, ',"charge":false,"charging_dock":1,"loading_speed":0}');
		fbClient.Publish(
            sTopic       := 'ChargingRequest',
            pPayload     := ADR(sSendCharging),
            nPayloadSize := LEN(sSendCharging),
            eQoS         := 0,
            bRetain      := FALSE,
            bQueue       := FALSE
         );
		 Charging := FALSE;
	END_IF
	
	IF (sMqttRECEIVE.sCmd.boCancelCharging OR sMqttRECEIVE.sCmd.boJobReset) AND fbClient.bConnected AND incharging_point2 = 1 AND (xinChargingPoint = 2) AND Charging THEN
		sSendCharging := CONCAT('{"robot":', INT_TO_STRING(Robot_Number));
		sSendCharging := CONCAT(sSendCharging, ',"charge":false,"charging_dock":2,"loading_speed":0}');
		fbClient.Publish(
            sTopic       := 'ChargingRequest',
            pPayload     := ADR(sSendCharging),
            nPayloadSize := LEN(sSendCharging),
            eQoS         := 0,
            bRetain      := FALSE,
            bQueue       := FALSE
         );
		 Charging := FALSE;
	END_IF

END_IF

// ============================================================
// Ausgabe
// ============================================================
ysDataToReceive := sMqttRECEIVE;

END_FUNCTION_BLOCK

// ---- POUs/HAWinoCore/001_MotorTask/Main_MotorTask.TcPOU
PROGRAM Main_MotorTask
VAR
	//////////////////////////////////////////////////////////////////////////////////////////////////////////
	// Variablen, die zur Synchronisation über das PAI (Prozessabbild) in den Task geladen werden.
	// -> Die Variablen werden von anderen Tasks gesetzt und müssen in den Task In/Outputs verknüpft werden
	//////////////////////////////////////////////////////////////////////////////////////////////////////////
	// Inputs für die Regelung
	n1fromMotor AT%I* : UINT; //Geschwindigkeit von der Motorklemme über den InfoData Kanal
	n2fromMotor AT%I* : UINT;
	n3fromMotor AT%I* : UINT;
	currentfromMotor1 AT %I* : UINT;	//Strom von der Motorklemme über den InfoData Kanal 2
	currentfromMotor2 AT %I* : UINT;
	currentfromMotor3 AT %I* : UINT;
	sliderGripper 		AT %I* : BOOL;

	//////////////////////////////////////////////////////////////////////////////////////////////////////////
	// Variablen werden zur Synchronisation über das PA-Q aus dem Task gesetzt.
	// -> Die Variablen werden von anderen Tasks gelesen.
	//////////////////////////////////////////////////////////////////////////////////////////////////////////

	// Freigabe der Motoren
	enableToMotor1 AT%Q*:BOOL:=FALSE;
	enableToMotor2 AT%Q*:BOOL:=FALSE;
	enableToMotor3 AT%Q*:BOOL:=FALSE;
	// Sollwerte der Motoren
	velocityToMotor1 AT%Q*:INT:=0;
	velocityToMotor2 AT%Q*:INT:=0;
	velocityToMotor3 AT%Q*:INT:=0;
	
	//////////////////////////////////////////////////////////////////////////////////////////////////////////
	// Taskinterne Inputs
	//////////////////////////////////////////////////////////////////////////////////////////////////////////
	// Wheel-Encoder Daten
	wheelEncoderLocalVx AT%I*		:LREAL;
	wheelEncoderLocalVy AT%I*		:LREAL;
	wheelEncoderLocalVtheta AT%I*	:LREAL;
	// Bumper Daten
	bumper AT%I* : BOOL;
	
	//////////////////////////////////////////////////////////////////////////////////////////////////////////
	// Lokale Variablen
	//////////////////////////////////////////////////////////////////////////////////////////////////////////
	
	// Übergabevariablen vom Lageregler zum Drehzahlregler
	vXCartesianToMotors 	:	LREAL;
	vYCartesianToMotors 	:	LREAL;
	vThetaCartesianToMotors :	LREAL;
	
	// Reglerdaten
	Motor1current: INT;
	Motor2current: INT;
	Motor3current: INT;

	velWheel1: LREAL;
	velWheel2: LREAL;
	velWheel3: LREAL;
	
	maxMotorRPM 			: INT 	:= 3600; 		// in rpm 
	maxKlemmeDrehzahlMessung: LREAL := 10000; 		// Bei Maximaldrehzahl zurückgegebener Drehzahlwert der Motorklemme
	rWheel 					: INT 	:= 40; 			// in mm
	ue						: LREAL := 0.0625; 		// Getriebeuebersetzung 
	cycletime 				: LREAL	:= 0.00033333; 	// Cycletime des Motortasks
	enableMotorControl		: BOOL  := TRUE;
	
	RobotIndex : INT := -1;
	
	DeltaWinkel : LREAL := 0.0;
	DeltaX : LREAL := 0.0;
	DeltaY : LREAL := 0.0;
	
	DeltaIn     : LREAL;
	DeltaLat    : LREAL;
	PosInOK     : BOOL;
	PosLatOK    : BOOL;
	
	WinkelOK: BOOL := FALSE;
	
	
	//////////////////////////////////////////////////////////////////////////////////////////////////////////
	// Instanzierung der FBs
	//////////////////////////////////////////////////////////////////////////////////////////////////////////

	FB_Drehzahlregler 	: FB_Drehzahlregler;	//Gilt für alle drei Motoren
	FB_Positionsregler 	: FB_Positionsregler;
	
	
	targetSpeed_World 	: sPosition;	// Geschwindigkeit in Weltkoordinaten
	targetSpeed_Robot	: sPosition;	// Geschwindigkeit in Roboterkoordinaten
	targetPos			: sPosition;	// Geschwindigkeitsvorgabe
	actualPos			: sPosition;	// Tatsächliche Position

	perfCamPos			: sPosition :=  (reWinkel := 0, reX := 0, reY := 0);	// vorherige Kamera Position

	VelAngle : LREAL; //Winkel in dem der Roboter fährt	
	IR_Distance : LREAL; // Minimaler Abstand des IR Sensors in Fahrtrichtung
	
	//Pseudofuzzy Parameter
	// Ersetzt die alten KPX_MIN/MAX etc. - umbenannt + gespiegelt für Lateral
	NILL        : LREAL := 0.0;
	
	KP_IN_MIN   : LREAL := 0.1;    // Einfahrrichtung KP minimum
	KP_IN_MAX   : LREAL := 3.0;    // Einfahrrichtung KP maximum
	KP_LAT_MIN  : LREAL := 1.0;    // Querrichtung KP minimum
	KP_LAT_MAX  : LREAL := 2.0;    // Querrichtung KP maximum
	KI_IN_MIN   : LREAL := 0.0;    // Einfahrrichtung KI disabled
	KI_IN_MAX   : LREAL := 0.25;    // Einfahrrichtung KI maximum
	
	// Berechnete Reglerwerte (generisch)
	KP_In       : LREAL;
	KP_Lat      : LREAL;
	KI_In       : LREAL;
	
	// Regler-Eingangswerte (gemappt auf X/Y des FB-Interfaces)
	KPX         : LREAL;
	KPY         : LREAL;
	KIX         : LREAL;
	KIY 		: LREAL;
	
	
	// Nil-Durchschaltung für gesperrte Achse
	vNILL_X     : LREAL := 0.0;    // Wird NILL zugewiesen wenn X gesperrt
	vNILL_Y     : LREAL := 0.0;    // Wird NILL zugewiesen wenn Y gesperrt
	
	ePocketOrientation : (ePocketX := 0, ePocketY := 1);
	
	f : LREAL;//Funktion für Übergang KIX und KPX
	
	wheelSpeed 			: WheelVelocity;
	

	diffPos		: sPosition;
	
	distanzeToRobot : LREAL;	// Abstandssensoren in mm
	
END_VAR

//Umrechung der Klemmenwerte
ACT_Drehzahlerfassung();

/////////////////////////////////////////////////////////////////////////////////////////////////////////
// Roboter-Positions-Bestimmung 
/////////////////////////////////////////////////////////////////////////////////////////////////////////
RobotIndex := Var_HAWIno.Robot_Number;
IF (RobotIndex < 1) OR (RobotIndex > 4) THEN
	// Falls außerhalb Bereich: Default auf 1 setzen 
	RobotIndex := -1;
ELSE

	wheelSpeed.wheel1  := -velWheel1;
	wheelSpeed.wheel2  := -velWheel2;
	wheelSpeed.wheel3  := -velWheel3;
	Beobachter(wheelSpeed := wheelSpeed, cameraData := Camera.cameraData, RobotIndex := RobotIndex, eastPos => actualPos);
	//enableMotorControl := FALSE;	
END_IF;

// Beste Positionsschätzung an Gruppe 2 übergeben
GVL_Datatransfer23.gvActualPosition		:= actualPos;


// Bei Bumper in den Fehler gehen
IF bumper THEN
	enableMotorControl := FALSE;
	GVL_Datatransfer23.inStatus := RobotStatus.fehler;	
END_IF

// Wenn keine Anfangsposition der Kamera gefunden wurde und der Roboter los fahren soll in den Fehlerzustand gehen
IF (actualPos.reX = 0 AND actualPos.reY = 0 AND  actualPos.reWinkel = 0) THEN
	IF GVL_Datatransfer23.inControl = RobotControl.vector OR  GVL_Datatransfer23.inControl = RobotControl.position THEN
		// enableMotorControl := FALSE;
		GVL_Datatransfer23.inStatus := RobotStatus.fehler;	
	END_IF
END_IF

//Gripper.closeGripperCommand := TRUE;
/////////////////////////////////////////////////////////////////////////////////////////////////////////
// Schrittkette
/////////////////////////////////////////////////////////////////////////////////////////////////////////
CASE GVL_Datatransfer23.inControl OF 
	RobotControl.idle:
		targetSpeed_Robot.reX		:= 0;
		targetSpeed_Robot.reY		:= 0;
		targetSpeed_Robot.reWinkel	:= 0;
		enableMotorControl := TRUE;
		GVL_Datatransfer23.inStatus	:= RobotStatus.betriebsbereit;

	RobotControl.stop:
		targetSpeed_Robot.reX		:= 0;
		targetSpeed_Robot.reY		:= 0;
		targetSpeed_Robot.reWinkel	:= 0;
		enableMotorControl := FALSE;
		GVL_Datatransfer23.inStatus	:= RobotStatus.fehler;
		
	RobotControl.reset:
		targetSpeed_Robot.reX		:= 0;
		targetSpeed_Robot.reY		:= 0;
		targetSpeed_Robot.reWinkel	:= 0;
		enableMotorControl := TRUE;
		GVL_Datatransfer23.inStatus	:= RobotStatus.betriebsbereit;
		
	/////////////////////////////////////////////////////////////////////////////////////////////////////////
	// Vector Regelung
	/////////////////////////////////////////////////////////////////////////////////////////////////////////
	RobotControl.vector:	
		// Geschwindigkeitsvektor von Gruppe 2 in Weltkoordinaten umrechnen
		targetSpeed_World.reX 	:= 		 GVL_Datatransfer23.gvFahrvektor.reGeschwindigkeit * COS(GVL_Datatransfer23.gvFahrvektor.reWinkel * PI /180.0);
		targetSpeed_World.reY 	:= (-1)* GVL_Datatransfer23.gvFahrvektor.reGeschwindigkeit * SIN(GVL_Datatransfer23.gvFahrvektor.reWinkel * PI /180.0);
		targetSpeed_World.reWinkel := 0;	// Zielwinkel in der Vectorregelung immer auf 0 setzen
		
		// Umrechnung der Geschwindigkeit von Welt in Roboterkoordinaten
		targetSpeed_Robot.reX 		:= targetSpeed_World.reX * COS(actualPos.reWinkel) - targetSpeed_World.reY * SIN(actualPos.reWinkel);
		targetSpeed_Robot.reY 		:= targetSpeed_World.reY * COS(actualPos.reWinkel) + targetSpeed_World.reX * SIN(actualPos.reWinkel);

		targetSpeed_Robot.reWinkel 	:= targetSpeed_World.reWinkel;	
		
		//targetSpeed_Robot.reX 		:= 0;
		//targetSpeed_Robot.reY 		:= 100;
		
		// VelAngle in Grad, 0°=+X, 90°=+Y, 180°=-X, 270°=-Y (CCW)
		VelAngle := ATAN2(targetSpeed_Robot.reY, targetSpeed_Robot.reX);

		// Negativen Bereich auf 0–360° normieren
		IF VelAngle < 0.0 THEN
    		VelAngle := VelAngle + 360.0;
		END_IF;
		
		IR_Distance := GetMinDistance(velAngle := VelAngle, tolerance := 45.0);
		
		IF IR_Distance < 100 THEN
			targetSpeed_Robot.reX 	:= 0;
			targetSpeed_Robot.reY 	:= 0;
		END_IF
		
		
	/////////////////////////////////////////////////////////////////////////////////////////////////////////
	// Positions Regelung
	/////////////////////////////////////////////////////////////////////////////////////////////////////////
	RobotControl.position:	
		targetPos.reX 		:= GVL_Datatransfer23.gvZielPosition.reX;
		targetPos.reY 		:= GVL_Datatransfer23.gvZielPosition.reY;
		targetPos.reWinkel	:= GVL_Datatransfer23.gvZielPosition.reWinkel* PI / 180.0;;
		// Prüfen ob Zielpositon erreicht
		

		// --- Pocket Orientation automatisch ermitteln ---
		IF ABS(ABS(targetPos.reWinkel) - (3.14159 / 2.0)) < 0.2 THEN
			ePocketOrientation := ePocketY;
		ELSE
			ePocketOrientation := ePocketX;
		END_IF
		
		// --- Deltas berechnen ---
		DeltaWinkel := ABS(actualPos.reWinkel) - ABS(targetPos.reWinkel);
		DeltaX      := ABS(actualPos.reX - targetPos.reX);
		DeltaY      := ABS(actualPos.reY - targetPos.reY);
		
		// Einfahr- und Querrichtung mappen
		IF ePocketOrientation = ePocketX THEN
			DeltaIn  := DeltaX;
			DeltaLat := DeltaY;
		ELSE
			DeltaIn  := DeltaY;
			DeltaLat := DeltaX;
		END_IF
		
		// --- Status-Flags ---
		IF ABS(DeltaWinkel) < 0.2   THEN WinkelOK := TRUE;  ELSE WinkelOK := FALSE;  END_IF
		IF DeltaIn          < 12    THEN PosInOK  := TRUE;  ELSE PosInOK  := FALSE;  END_IF
		IF DeltaLat         < 2     THEN PosLatOK := TRUE;  ELSE PosLatOK := FALSE;  END_IF		
		
		// --- Adaptive Verstärkung (Einfahrrichtung) ---
		f := DeltaIn / 100.0;
		IF f > 1 THEN f := 1; END_IF
		IF f < 0 THEN f := 0; END_IF
		
		IF DeltaIn < 35 THEN
			KP_In := 0;
		ELSE
			KP_In := KP_IN_MIN + f * (KP_IN_MAX - KP_IN_MIN);
		END_IF
		
		IF DeltaIn > 100 THEN
			KI_In := 0;
		ELSE
			KI_In := KI_IN_MAX - f * (KI_IN_MAX - KI_IN_MIN);
		END_IF
		
		KP_Lat := KP_LAT_MAX;
		
		// --- KPX/KPY/KIX/KIY auf FB-Interface mappen ---
		IF ePocketOrientation = ePocketX THEN
			KPX := KP_In;
			KPY := KP_Lat;
			KIX := KI_In;
			KIY := NILL;     // Lateral-Integral nicht benötigt
		ELSE
			KPX := KP_Lat;   // FB-X ist Querrichtung
			KPY := KP_In;    // FB-Y ist Einfahrrichtung
			KIX := NILL;     // Lateral-Integral nicht benötigt
			KIY := KI_In;    // Integral liegt jetzt auf Y
		END_IF
		
		// --- Regleraufrufe ---
		
		// 1. Winkel ausrichten
		IF (WinkelOK = FALSE) THEN
			FB_Positionsregler(targetPos := targetPos, actualPos := actualPos,
								vXCartesianToMotors     => targetSpeed_Robot.reX,
								vYCartesianToMotors     => targetSpeed_Robot.reY,
								vThetaCartesianToMotors => targetSpeed_Robot.reWinkel);
								targetSpeed_Robot.reX := 0;
								targetSpeed_Robot.reY := 0;
			GVL_Datatransfer23.inStatus := RobotStatus.laufend;
		
		// 2. Nah an Tasche aber lateral daneben: nur Querrichtung
		ELSIF (DeltaLat > 5 AND DeltaIn < 20) THEN
			IF ePocketOrientation = ePocketX THEN
				FB_Positionsregler(targetPos := targetPos, actualPos := actualPos,
									KPX := NILL, KPY := KPY, KIX := NILL, KIY := NILL,
									vXCartesianToMotors     => targetSpeed_Robot.reX,
									vYCartesianToMotors     => targetSpeed_Robot.reY,
									vThetaCartesianToMotors => targetSpeed_Robot.reWinkel);
									targetSpeed_Robot.reX := 0;
			ELSE
				FB_Positionsregler(targetPos := targetPos, actualPos := actualPos,
									KPX := KPX, KPY := NILL, KIX := NILL, KIY := NILL,
									vXCartesianToMotors     => targetSpeed_Robot.reX,
									vYCartesianToMotors     => targetSpeed_Robot.reY,
									vThetaCartesianToMotors => targetSpeed_Robot.reWinkel);
									targetSpeed_Robot.reY := 0;
			END_IF
			GVL_Datatransfer23.inStatus := RobotStatus.laufend;
		
